LIN {X 0,Y 467.077,Z 400.09,A -85,B 0,C 180,E1 -7772.581,E2 -7772.581} C_VEL
LIN {X 0,Y 466.879,Z 403.998,A -85,B 0,C 180,E1 -7774.113,E2 -7774.113} C_VEL
LIN {X 0,Y 466.736,Z 406.492,A -85,B 0,C 180,E1 -7775.597,E2 -7775.597} C_VEL
LIN {X 0,Y 466.664,Z 407.771,A -85,B 0,C 180,E1 -7777.042,E2 -7777.042} C_VEL
LIN {X 0,Y 466.681,Z 407.948,A -85,B 0,C 180,E1 -7778.454,E2 -7778.454} C_VEL
LIN {X 0,Y 466.711,Z 407.112,A -85,B 0,C 180,E1 -7779.826,E2 -7779.826} C_VEL
LIN {X 0,Y 466.814,Z 404.771,A -85,B 0,C 180,E1 -7781.486,E2 -7781.486} C_VEL
LIN {X 0,Y 467.044,Z 400.686,A -85,B 0,C 180,E1 -7783.189,E2 -7783.189} C_VEL
LIN {X 0,Y 467.228,Z 395.648,A -85,B 0,C 180,E1 -7784.685,E2 -7784.685} C_VEL
LIN {X 0,Y 467.456,Z 388.922,A -85,B 0,C 180,E1 -7786.192,E2 -7786.192} C_VEL
LIN {X 0,Y 467.852,Z 381.695,A -85,B 0,C 180,E1 -7787.469,E2 -7787.469} C_VEL
LIN {X 0,Y 468.223,Z 373.379,A -85,B 0,C 180,E1 -7788.666,E2 -7788.666} C_VEL
LIN {X 0,Y 468.647,Z 364.557,A -85,B 0,C 180,E1 -7789.705,E2 -7789.705} C_VEL
LIN {X 0,Y 469.155,Z 353.711,A -85,B 0,C 180,E1 -7790.734,E2 -7790.734} C_VEL
LIN {X 0,Y 469.63,Z 342.193,A -85,B 0,C 180,E1 -7791.607,E2 -7791.607} C_VEL
LIN {X 0,Y 470.092,Z 330.037,A -85,B 0,C 180,E1 -7792.316,E2 -7792.316} C_VEL
LIN {X 0,Y 470.223,Z 319.07,A -85,B 0,C 180,E1 -7792.805,E2 -7792.805} C_VEL
LIN {X 0,Y 466.983,Z 306.035,A -85,B 0,C 180,E1 -7793.324,E2 -7793.324} C_VEL
LIN {X 0,Y 466.864,Z 305.117,A -85,B 0,C 180,E1 -7793.38,E2 -7793.38} C_VEL
LIN {X 0,Y 466.879,Z 302.169,A -85,B 0,C 180,E1 -7796.153,E2 -7796.153} C_VEL
LIN {X 0,Y 466.906,Z 298.871,A -85,B 0,C 180,E1 -7799.302,E2 -7799.302} C_VEL
LIN {X 0,Y 466.963,Z 296.873,A -85,B 0,C 180,E1 -7801.209,E2 -7801.209} C_VEL
LIN {X 0,Y 467.055,Z 296.311,A -85,B 0,C 180,E1 -7802.598,E2 -7802.598} C_VEL
LIN {X 0,Y 467.101,Z 296.304,A -85,B 0,C 180,E1 -7803.04,E2 -7803.04} C_VEL
LIN {X 0,Y 466.541,Z 296.375,A -85,B 0,C 180,E1 -7803.76,E2 -7803.76} C_VEL
LIN {X 0,Y 463.844,Z 296.712,A -85,B 0,C 180,E1 -7804.934,E2 -7804.934} C_VEL
LIN {X 0,Y 461.52,Z 297,A -85,B 0,C 180,E1 -7805.88,E2 -7805.88} C_VEL
LIN {X 0,Y 460.523,Z 297.122,A -85,B 0,C 180,E1 -7806.609,E2 -7806.609} C_VEL
LIN {X 0,Y 460.446,Z 297.13,A -85,B 0,C 180,E1 -7806.856,E2 -7806.856} C_VEL
LIN {X 0,Y 460.552,Z 297.12,A -85,B 0,C 180,E1 -7809.453,E2 -7809.453} C_VEL
LIN {X 0,Y 460.549,Z 297.118,A -85,B 0,C 180,E1 -7812.23,E2 -7812.23} C_VEL
LIN {X 0,Y 460.566,Z 297.118,A -85,B 0,C 180,E1 -7814.965,E2 -7814.965} C_VEL
LIN {X 0,Y 460.611,Z 297.11,A -85,B 0,C 180,E1 -7818.559,E2 -7818.559} C_VEL
LIN {X 0,Y 460.668,Z 297.101,A -85,B 0,C 180,E1 -7822.108,E2 -7822.108} C_VEL
LIN {X 0,Y 460.691,Z 297.101,A -85,B 0,C 180,E1 -7824.748,E2 -7824.748} C_VEL
LIN {X 0,Y 460.801,Z 297.086,A -85,B 0,C 180,E1 -7827.377,E2 -7827.377} C_VEL
LIN {X 0,Y 460.854,Z 297.078,A -85,B 0,C 180,E1 -7830,E2 -7830} C_VEL
LIN {X 0,Y 460.826,Z 297.084,A -85,B 0,C 180,E1 -7832.622,E2 -7832.622} C_VEL
LIN {X 0,Y 460.685,Z 297.102,A -85,B 0,C 180,E1 -7836.13,E2 -7836.13} C_VEL
LIN {X 0,Y 460.628,Z 297.109,A -85,B 0,C 180,E1 -7838.776,E2 -7838.776} C_VEL
LIN {X 0,Y 460.615,Z 297.112,A -85,B 0,C 180,E1 -7842.445,E2 -7842.445} C_VEL
LIN {X 0,Y 460.602,Z 297.111,A -85,B 0,C 180,E1 -7845.998,E2 -7845.998} C_VEL
LIN {X 0,Y 460.569,Z 297.114,A -85,B 0,C 180,E1 -7849.616,E2 -7849.616} C_VEL
LIN {X 0,Y 460.513,Z 297.123,A -85,B 0,C 180,E1 -7852.429,E2 -7852.429} C_VEL
LIN {X 0,Y 460.57,Z 297.117,A -85,B 0,C 180,E1 -7855.802,E2 -7855.802} C_VEL
LIN {X 0,Y 460.552,Z 297.119,A -85,B 0,C 180,E1 -7858.233,E2 -7858.233} C_VEL
LIN {X 0,Y 460.521,Z 297.12,A -85,B 0,C 180,E1 -7861.283,E2 -7861.283} C_VEL
LIN {X 0,Y 460.525,Z 297.122,A -85,B 0,C 180,E1 -7864.504,E2 -7864.504} C_VEL
LIN {X 0,Y 460.503,Z 297.125,A -85,B 0,C 180,E1 -7867.623,E2 -7867.623} C_VEL
LIN {X 0,Y 460.544,Z 297.119,A -85,B 0,C 180,E1 -7870.27,E2 -7870.27} C_VEL
LIN {X 0,Y 460.498,Z 297.124,A -85,B 0,C 180,E1 -7873.376,E2 -7873.376} C_VEL
LIN {X 0,Y 460.501,Z 297.123,A -85,B 0,C 180,E1 -7876.625,E2 -7876.625} C_VEL
LIN {X 0,Y 460.545,Z 297.119,A -85,B 0,C 180,E1 -7879.731,E2 -7879.731} C_VEL
LIN {X 0,Y 460.503,Z 297.123,A -85,B 0,C 180,E1 -7882.524,E2 -7882.524} C_VEL
LIN {X 0,Y 460.54,Z 297.122,A -85,B 0,C 180,E1 -7885.623,E2 -7885.623} C_VEL
LIN {X 0,Y 460.54,Z 297.119,A -85,B 0,C 180,E1 -7888.745,E2 -7888.745} C_VEL
LIN {X 0,Y 460.581,Z 297.114,A -85,B 0,C 180,E1 -7892.255,E2 -7892.255} C_VEL
LIN {X 0,Y 460.529,Z 297.121,A -85,B 0,C 180,E1 -7895.667,E2 -7895.667} C_VEL
LIN {X 0,Y 460.525,Z 297.12,A -85,B 0,C 180,E1 -7898.578,E2 -7898.578} C_VEL
LIN {X 0,Y 460.59,Z 297.115,A -85,B 0,C 180,E1 -7901.311,E2 -7901.311} C_VEL
LIN {X 0,Y 460.609,Z 297.11,A -85,B 0,C 180,E1 -7904.059,E2 -7904.059} C_VEL
LIN {X 0,Y 460.614,Z 297.111,A -85,B 0,C 180,E1 -7907.666,E2 -7907.666} C_VEL
LIN {X 0,Y 460.624,Z 297.109,A -85,B 0,C 180,E1 -7911.224,E2 -7911.224} C_VEL
LIN {X 0,Y 460.712,Z 297.096,A -85,B 0,C 180,E1 -7913.87,E2 -7913.87} C_VEL
LIN {X 0,Y 460.798,Z 297.087,A -85,B 0,C 180,E1 -7917.378,E2 -7917.378} C_VEL
LIN {X 0,Y 460.857,Z 297.079,A -85,B 0,C 180,E1 -7920,E2 -7920} C_VEL
LIN {X 0,Y 460.793,Z 297.09,A -85,B 0,C 180,E1 -7922.623,E2 -7922.623} C_VEL
LIN {X 0,Y 460.688,Z 297.1,A -85,B 0,C 180,E1 -7926.13,E2 -7926.13} C_VEL
LIN {X 0,Y 460.623,Z 297.11,A -85,B 0,C 180,E1 -7928.776,E2 -7928.776} C_VEL
LIN {X 0,Y 460.619,Z 297.11,A -85,B 0,C 180,E1 -7932.445,E2 -7932.445} C_VEL
LIN {X 0,Y 460.605,Z 297.111,A -85,B 0,C 180,E1 -7935.998,E2 -7935.998} C_VEL
LIN {X 0,Y 460.572,Z 297.115,A -85,B 0,C 180,E1 -7939.616,E2 -7939.616} C_VEL
LIN {X 0,Y 460.515,Z 297.123,A -85,B 0,C 180,E1 -7942.429,E2 -7942.429} C_VEL
LIN {X 0,Y 460.552,Z 297.117,A -85,B 0,C 180,E1 -7945.797,E2 -7945.797} C_VEL
LIN {X 0,Y 460.531,Z 297.121,A -85,B 0,C 180,E1 -7948.235,E2 -7948.235} C_VEL
LIN {X 0,Y 460.525,Z 297.121,A -85,B 0,C 180,E1 -7951.283,E2 -7951.283} C_VEL
LIN {X 0,Y 460.535,Z 297.12,A -85,B 0,C 180,E1 -7954.505,E2 -7954.505} C_VEL
LIN {X 0,Y 460.505,Z 297.123,A -85,B 0,C 180,E1 -7957.623,E2 -7957.623} C_VEL
LIN {X 0,Y 460.54,Z 297.121,A -85,B 0,C 180,E1 -7960.268,E2 -7960.268} C_VEL
LIN {X 0,Y 460.512,Z 297.124,A -85,B 0,C 180,E1 -7963.374,E2 -7963.374} C_VEL
LIN {X 0,Y 460.512,Z 297.121,A -85,B 0,C 180,E1 -7966.626,E2 -7966.626} C_VEL
LIN {X 0,Y 460.571,Z 297.238,A -85,B 0,C 180,E1 -7969.444,E2 -7969.444} C_VEL
LIN {X 0,Y 462.242,Z 306.265,A -85,B 0,C 180,E1 -7973.089,E2 -7973.089} C_VEL
LIN {X 0,Y 462.399,Z 310.595,A -85,B 0,C 180,E1 -7974.72,E2 -7974.72} C_VEL
LIN {X 0,Y 461.883,Z 319.246,A -85,B 0,C 180,E1 -7977.821,E2 -7977.821} C_VEL
LIN {X 0,Y 461.323,Z 329.384,A -85,B 0,C 180,E1 -7981.322,E2 -7981.322} C_VEL
LIN {X 0,Y 460.86,Z 339.544,A -85,B 0,C 180,E1 -7984.723,E2 -7984.723} C_VEL
LIN {X 0,Y 460.428,Z 349.692,A -85,B 0,C 180,E1 -7988.039,E2 -7988.039} C_VEL
LIN {X 0,Y 460.203,Z 359.887,A -85,B 0,C 180,E1 -7991.294,E2 -7991.294} C_VEL
LIN {X 0,Y 459.948,Z 369.672,A -85,B 0,C 180,E1 -7994.36,E2 -7994.36} C_VEL
LIN {X 0,Y 461.927,Z 384.605,A -85,B 0,C 180,E1 -7994.838,E2 -7994.838} C_VEL
LIN {X 0,Y 462.821,Z 394.468,A -85,B 0,C 180,E1 -7995.265,E2 -7995.265} C_VEL
LIN {X 0,Y 462.305,Z 406.889,A -85,B 0,C 180,E1 -7995.922,E2 -7995.922} C_VEL
LIN {X 0,Y 461.662,Z 419.477,A -85,B 0,C 180,E1 -7996.8,E2 -7996.8} C_VEL
LIN {X 0,Y 461.143,Z 430.593,A -85,B 0,C 180,E1 -7997.792,E2 -7997.792} C_VEL
LIN {X 0,Y 460.751,Z 439.624,A -85,B 0,C 180,E1 -7998.786,E2 -7998.786} C_VEL
LIN {X 0,Y 460.265,Z 449.421,A -85,B 0,C 180,E1 -8000.109,E2 -8000.109} C_VEL
LIN {X 0,Y 459.999,Z 457.267,A -85,B 0,C 180,E1 -8001.433,E2 -8001.433} C_VEL
LIN {X 0,Y 459.777,Z 464.466,A -85,B 0,C 180,E1 -8002.976,E2 -8002.976} C_VEL
LIN {X 0,Y 459.718,Z 469.266,A -85,B 0,C 180,E1 -8004.297,E2 -8004.297} C_VEL
LIN {X 0,Y 459.604,Z 472.924,A -85,B 0,C 180,E1 -8005.615,E2 -8005.615} C_VEL
LIN {X 0,Y 459.686,Z 474.819,A -85,B 0,C 180,E1 -8006.494,E2 -8006.494} C_VEL
LIN {X 0,Y 459.689,Z 476.233,A -85,B 0,C 180,E1 -8007.371,E2 -8007.371} C_VEL
LIN {X 0,Y 459.637,Z 477.228,A -85,B 0,C 180,E1 -8008.248,E2 -8008.248} C_VEL
LIN {X 0,Y 459.554,Z 478.027,A -85,B 0,C 180,E1 -8010,E2 -8010} C_VEL
LIN {X 0,Y 459.567,Z 477.788,A -85,B 0,C 180,E1 -8010.876,E2 -8010.876} C_VEL
LIN {X 0,Y 459.638,Z 477.151,A -85,B 0,C 180,E1 -8011.752,E2 -8011.752} C_VEL
LIN {X 0,Y 459.705,Z 476.116,A -85,B 0,C 180,E1 -8012.629,E2 -8012.629} C_VEL
LIN {X 0,Y 459.699,Z 474.666,A -85,B 0,C 180,E1 -8013.506,E2 -8013.506} C_VEL
LIN {X 0,Y 459.637,Z 471.625,A -85,B 0,C 180,E1 -8014.824,E2 -8014.824} C_VEL
LIN {X 0,Y 459.699,Z 467.531,A -85,B 0,C 180,E1 -8016.144,E2 -8016.144} C_VEL
LIN {X 0,Y 459.865,Z 461.251,A -85,B 0,C 180,E1 -8017.685,E2 -8017.685} C_VEL
LIN {X 0,Y 460.063,Z 454.403,A -85,B 0,C 180,E1 -8019.009,E2 -8019.009} C_VEL
LIN {X 0,Y 460.383,Z 445.938,A -85,B 0,C 180,E1 -8020.333,E2 -8020.333} C_VEL
LIN {X 0,Y 460.854,Z 437.273,A -85,B 0,C 180,E1 -8021.435,E2 -8021.435} C_VEL
LIN {X 0,Y 461.274,Z 427.652,A -85,B 0,C 180,E1 -8022.441,E2 -8022.441} C_VEL
LIN {X 0,Y 461.754,Z 416.085,A -85,B 0,C 180,E1 -8023.421,E2 -8023.421} C_VEL
LIN {X 0,Y 462.357,Z 404.606,A -85,B 0,C 180,E1 -8024.188,E2 -8024.188} C_VEL
LIN {X 0,Y 462.843,Z 392.852,A -85,B 0,C 180,E1 -8024.791,E2 -8024.791} C_VEL
LIN {X 0,Y 461.404,Z 379.556,A -85,B 0,C 180,E1 -8025.344,E2 -8025.344} C_VEL
LIN {X 0,Y 459.918,Z 368.362,A -85,B 0,C 180,E1 -8025.697,E2 -8025.697} C_VEL
LIN {X 0,Y 460.106,Z 358.542,A -85,B 0,C 180,E1 -8028.731,E2 -8028.731} C_VEL
LIN {X 0,Y 460.328,Z 349.752,A -85,B 0,C 180,E1 -8031.495,E2 -8031.495} C_VEL
LIN {X 0,Y 460.62,Z 339.486,A -85,B 0,C 180,E1 -8034.809,E2 -8034.809} C_VEL
LIN {X 0,Y 461.018,Z 330.389,A -85,B 0,C 180,E1 -8037.848,E2 -8037.848} C_VEL
LIN {X 0,Y 461.574,Z 319.93,A -85,B 0,C 180,E1 -8041.497,E2 -8041.497} C_VEL
LIN {X 0,Y 462.185,Z 311,A -85,B 0,C 180,E1 -8044.802,E2 -8044.802} C_VEL
LIN {X 0,Y 462.234,Z 307.021,A -85,B 0,C 180,E1 -8046.369,E2 -8046.369} C_VEL
LIN {X 0,Y 461.377,Z 301.675,A -85,B 0,C 180,E1 -8048.649,E2 -8048.649} C_VEL
LIN {X 0,Y 460.566,Z 297.118,A -85,B 0,C 180,E1 -8050.808,E2 -8050.808} C_VEL
LIN {X 0,Y 460.516,Z 297.127,A -85,B 0,C 180,E1 -8054.17,E2 -8054.17} C_VEL
LIN {X 0,Y 460.517,Z 297.127,A -85,B 0,C 180,E1 -8057.1,E2 -8057.1} C_VEL
LIN {X 0,Y 460.537,Z 297.123,A -85,B 0,C 180,E1 -8060.138,E2 -8060.138} C_VEL
LIN {X 0,Y 460.481,Z 297.127,A -85,B 0,C 180,E1 -8063.471,E2 -8063.471} C_VEL
LIN {X 0,Y 460.534,Z 297.121,A -85,B 0,C 180,E1 -8066.675,E2 -8066.675} C_VEL
LIN {X 0,Y 460.516,Z 297.123,A -85,B 0,C 180,E1 -8069.76,E2 -8069.76} C_VEL
LIN {X 0,Y 460.584,Z 297.114,A -85,B 0,C 180,E1 -8072.757,E2 -8072.757} C_VEL
LIN {X 0,Y 460.547,Z 297.117,A -85,B 0,C 180,E1 -8075.668,E2 -8075.668} C_VEL
LIN {X 0,Y 460.526,Z 297.122,A -85,B 0,C 180,E1 -8078.578,E2 -8078.578} C_VEL
LIN {X 0,Y 460.591,Z 297.114,A -85,B 0,C 180,E1 -8081.311,E2 -8081.311} C_VEL
LIN {X 0,Y 460.609,Z 297.111,A -85,B 0,C 180,E1 -8084.059,E2 -8084.059} C_VEL
LIN {X 0,Y 460.615,Z 297.111,A -85,B 0,C 180,E1 -8087.666,E2 -8087.666} C_VEL
LIN {X 0,Y 460.624,Z 297.109,A -85,B 0,C 180,E1 -8091.224,E2 -8091.224} C_VEL
LIN {X 0,Y 460.688,Z 297.101,A -85,B 0,C 180,E1 -8093.87,E2 -8093.87} C_VEL
LIN {X 0,Y 460.805,Z 297.087,A -85,B 0,C 180,E1 -8097.377,E2 -8097.377} C_VEL
LIN {X 0,Y 460.859,Z 297.082,A -85,B 0,C 180,E1 -8100,E2 -8100} C_VEL
LIN {X 0,Y 460.83,Z 297.084,A -85,B 0,C 180,E1 -8102.622,E2 -8102.622} C_VEL
LIN {X 0,Y 460.691,Z 297.103,A -85,B 0,C 180,E1 -8106.13,E2 -8106.13} C_VEL
LIN {X 0,Y 460.567,Z 297.118,A -85,B 0,C 180,E1 -8108.777,E2 -8108.777} C_VEL
LIN {X 0,Y 460.334,Z 297.148,A -85,B 0,C 180,E1 -8111.448,E2 -8111.448} C_VEL
LIN {X 0,Y 460.26,Z 297.442,A -85,B 0,C 180,E1 -8112.344,E2 -8112.344} C_VEL
LIN {X 0,Y 460.14,Z 300.675,A -85,B 0,C 180,E1 -8115.794,E2 -8115.794} C_VEL
LIN {X 0,Y 460.01,Z 303.468,A -85,B 0,C 180,E1 -8118.713,E2 -8118.713} C_VEL
LIN {X 0,Y 459.961,Z 306.142,A -85,B 0,C 180,E1 -8121.513,E2 -8121.513} C_VEL
LIN {X 0,Y 459.936,Z 307.052,A -85,B 0,C 180,E1 -8122.458,E2 -8122.458} C_VEL
LIN {X 0,Y 463.555,Z 320.766,A -85,B 0,C 180,E1 -8123.038,E2 -8123.038} C_VEL
LIN {X 0,Y 463.367,Z 332.506,A -85,B 0,C 180,E1 -8123.58,E2 -8123.58} C_VEL
LIN {X 0,Y 462.938,Z 343.442,A -85,B 0,C 180,E1 -8124.24,E2 -8124.24} C_VEL
LIN {X 0,Y 462.404,Z 354.286,A -85,B 0,C 180,E1 -8125.071,E2 -8125.071} C_VEL
LIN {X 0,Y 461.861,Z 365.295,A -85,B 0,C 180,E1 -8126.13,E2 -8126.13} C_VEL
LIN {X 0,Y 461.396,Z 374.199,A -85,B 0,C 180,E1 -8127.191,E2 -8127.191} C_VEL
LIN {X 0,Y 460.985,Z 382.758,A -85,B 0,C 180,E1 -8128.452,E2 -8128.452} C_VEL
LIN {X 0,Y 460.529,Z 390.5,A -85,B 0,C 180,E1 -8129.87,E2 -8129.87} C_VEL
LIN {X 0,Y 460.249,Z 396.54,A -85,B 0,C 180,E1 -8131.277,E2 -8131.277} C_VEL
LIN {X 0,Y 459.98,Z 401.571,A -85,B 0,C 180,E1 -8132.823,E2 -8132.823} C_VEL
LIN {X 0,Y 459.778,Z 405.325,A -85,B 0,C 180,E1 -8134.442,E2 -8134.442} C_VEL
LIN {X 0,Y 459.63,Z 407.418,A -85,B 0,C 180,E1 -8135.864,E2 -8135.864} C_VEL
LIN {X 0,Y 459.584,Z 408.46,A -85,B 0,C 180,E1 -8137.326,E2 -8137.326} C_VEL
LIN {X 0,Y 459.622,Z 408.377,A -85,B 0,C 180,E1 -8138.823,E2 -8138.823} C_VEL
LIN {X 0,Y 459.64,Z 407.369,A -85,B 0,C 180,E1 -8140.136,E2 -8140.136} C_VEL
LIN {X 0,Y 459.755,Z 405.367,A -85,B 0,C 180,E1 -8141.493,E2 -8141.493} C_VEL
LIN {X 0,Y 459.925,Z 402.426,A -85,B 0,C 180,E1 -8142.821,E2 -8142.821} C_VEL
LIN {X 0,Y 460.064,Z 398.573,A -85,B 0,C 180,E1 -8144.112,E2 -8144.112} C_VEL
LIN {X 0,Y 460.33,Z 392.861,A -85,B 0,C 180,E1 -8145.58,E2 -8145.58} C_VEL
LIN {X 0,Y 460.653,Z 385.313,A -85,B 0,C 180,E1 -8147.081,E2 -8147.081} C_VEL
LIN {X 0,Y 461.073,Z 377.507,A -85,B 0,C 180,E1 -8148.322,E2 -8148.322} C_VEL
LIN {X 0,Y 461.504,Z 369.477,A -85,B 0,C 180,E1 -8149.37,E2 -8149.37} C_VEL
LIN {X 0,Y 462.003,Z 359.381,A -85,B 0,C 180,E1 -8150.446,E2 -8150.446} C_VEL
LIN {X 0,Y 462.448,Z 349.392,A -85,B 0,C 180,E1 -8151.311,E2 -8151.311} C_VEL
LIN {X 0,Y 462.977,Z 337.6,A -85,B 0,C 180,E1 -8152.126,E2 -8152.126} C_VEL
LIN {X 0,Y 463.387,Z 326.476,A -85,B 0,C 180,E1 -8152.719,E2 -8152.719} C_VEL
LIN {X 0,Y 463.353,Z 320.314,A -85,B 0,C 180,E1 -8152.989,E2 -8152.989} C_VEL
LIN {X 0,Y 460.088,Z 307.047,A -85,B 0,C 180,E1 -8153.532,E2 -8153.532} C_VEL
LIN {X 0,Y 459.793,Z 305.583,A -85,B 0,C 180,E1 -8153.602,E2 -8153.602} C_VEL
LIN {X 0,Y 459.829,Z 301.774,A -85,B 0,C 180,E1 -8157.205,E2 -8157.205} C_VEL
LIN {X 0,Y 459.862,Z 298.238,A -85,B 0,C 180,E1 -8160.589,E2 -8160.589} C_VEL
LIN {X 0,Y 459.918,Z 297.202,A -85,B 0,C 180,E1 -8161.724,E2 -8161.724} C_VEL
LIN {X 0,Y 460.274,Z 297.154,A -85,B 0,C 180,E1 -8164.688,E2 -8164.688} C_VEL
LIN {X 0,Y 460.446,Z 297.13,A -85,B 0,C 180,E1 -8166.856,E2 -8166.856} C_VEL
LIN {X 0,Y 459.791,Z 297.213,A -85,B 0,C 180,E1 -8167.586,E2 -8167.586} C_VEL
LIN {X 0,Y 456.961,Z 297.565,A -85,B 0,C 180,E1 -8168.773,E2 -8168.773} C_VEL
LIN {X 0,Y 454.577,Z 297.861,A -85,B 0,C 180,E1 -8169.73,E2 -8169.73} C_VEL
LIN {X 0,Y 453.574,Z 297.985,A -85,B 0,C 180,E1 -8170.47,E2 -8170.47} C_VEL
LIN {X 0,Y 453.503,Z 297.995,A -85,B 0,C 180,E1 -8170.72,E2 -8170.72} C_VEL
LIN {X 0,Y 453.57,Z 297.985,A -85,B 0,C 180,E1 -8173.88,E2 -8173.88} C_VEL
LIN {X 0,Y 453.565,Z 297.988,A -85,B 0,C 180,E1 -8177.471,E2 -8177.471} C_VEL
LIN {X 0,Y 453.592,Z 297.986,A -85,B 0,C 180,E1 -8181.087,E2 -8181.087} C_VEL
LIN {X 0,Y 453.652,Z 297.977,A -85,B 0,C 180,E1 -8183.774,E2 -8183.774} C_VEL
LIN {X 0,Y 453.745,Z 297.965,A -85,B 0,C 180,E1 -8187.337,E2 -8187.337} C_VEL
LIN {X 0,Y 453.824,Z 297.954,A -85,B 0,C 180,E1 -8190,E2 -8190} C_VEL
LIN {X 0,Y 453.767,Z 297.963,A -85,B 0,C 180,E1 -8192.663,E2 -8192.663} C_VEL
LIN {X 0,Y 453.651,Z 297.978,A -85,B 0,C 180,E1 -8196.226,E2 -8196.226} C_VEL
LIN {X 0,Y 453.592,Z 297.985,A -85,B 0,C 180,E1 -8198.913,E2 -8198.913} C_VEL
LIN {X 0,Y 453.565,Z 297.99,A -85,B 0,C 180,E1 -8202.529,E2 -8202.529} C_VEL
LIN {X 0,Y 453.545,Z 297.992,A -85,B 0,C 180,E1 -8206.196,E2 -8206.196} C_VEL
LIN {X 0,Y 453.517,Z 297.993,A -85,B 0,C 180,E1 -8209.039,E2 -8209.039} C_VEL
LIN {X 0,Y 453.478,Z 298,A -85,B 0,C 180,E1 -8211.836,E2 -8211.836} C_VEL
LIN {X 0,Y 453.516,Z 297.993,A -85,B 0,C 180,E1 -8214.735,E2 -8214.735} C_VEL
LIN {X 0,Y 453.533,Z 297.993,A -85,B 0,C 180,E1 -8217.96,E2 -8217.96} C_VEL
LIN {X 0,Y 453.466,Z 297.999,A -85,B 0,C 180,E1 -8221.525,E2 -8221.525} C_VEL
LIN {X 0,Y 453.484,Z 297.998,A -85,B 0,C 180,E1 -8224.777,E2 -8224.777} C_VEL
LIN {X 0,Y 453.467,Z 298.002,A -85,B 0,C 180,E1 -8228.312,E2 -8228.312} C_VEL
LIN {X 0,Y 453.496,Z 297.996,A -85,B 0,C 180,E1 -8230.609,E2 -8230.609} C_VEL
LIN {X 0,Y 453.455,Z 298.001,A -85,B 0,C 180,E1 -8233.244,E2 -8233.244} C_VEL
LIN {X 0,Y 453.466,Z 298.001,A -85,B 0,C 180,E1 -8235.779,E2 -8235.779} C_VEL
LIN {X 0,Y 453.482,Z 297.998,A -85,B 0,C 180,E1 -8238.21,E2 -8238.21} C_VEL
LIN {X 0,Y 453.518,Z 297.993,A -85,B 0,C 180,E1 -8240.79,E2 -8240.79} C_VEL
LIN {X 0,Y 453.457,Z 298.002,A -85,B 0,C 180,E1 -8243.917,E2 -8243.917} C_VEL
LIN {X 0,Y 453.482,Z 298,A -85,B 0,C 180,E1 -8247.151,E2 -8247.151} C_VEL
LIN {X 0,Y 453.478,Z 297.997,A -85,B 0,C 180,E1 -8250.269,E2 -8250.269} C_VEL
LIN {X 0,Y 453.492,Z 297.998,A -85,B 0,C 180,E1 -8253.293,E2 -8253.293} C_VEL
LIN {X 0,Y 453.498,Z 297.996,A -85,B 0,C 180,E1 -8256.239,E2 -8256.239} C_VEL
LIN {X 0,Y 453.487,Z 297.999,A -85,B 0,C 180,E1 -8259.118,E2 -8259.118} C_VEL
LIN {X 0,Y 453.507,Z 297.994,A -85,B 0,C 180,E1 -8261.944,E2 -8261.944} C_VEL
LIN {X 0,Y 453.544,Z 297.99,A -85,B 0,C 180,E1 -8264.727,E2 -8264.727} C_VEL
LIN {X 0,Y 453.564,Z 297.988,A -85,B 0,C 180,E1 -8268.379,E2 -8268.379} C_VEL
LIN {X 0,Y 453.59,Z 297.986,A -85,B 0,C 180,E1 -8271.087,E2 -8271.087} C_VEL
LIN {X 0,Y 453.678,Z 297.972,A -85,B 0,C 180,E1 -8273.775,E2 -8273.775} C_VEL
LIN {X 0,Y 453.741,Z 297.966,A -85,B 0,C 180,E1 -8277.337,E2 -8277.337} C_VEL
LIN {X 0,Y 453.826,Z 297.955,A -85,B 0,C 180,E1 -8280,E2 -8280} C_VEL
LIN {X 0,Y 453.737,Z 297.968,A -85,B 0,C 180,E1 -8282.663,E2 -8282.663} C_VEL
LIN {X 0,Y 453.654,Z 297.976,A -85,B 0,C 180,E1 -8286.226,E2 -8286.226} C_VEL
LIN {X 0,Y 453.589,Z 297.987,A -85,B 0,C 180,E1 -8288.914,E2 -8288.914} C_VEL
LIN {X 0,Y 453.569,Z 297.988,A -85,B 0,C 180,E1 -8292.529,E2 -8292.529} C_VEL
LIN {X 0,Y 453.549,Z 297.99,A -85,B 0,C 180,E1 -8296.196,E2 -8296.196} C_VEL
LIN {X 0,Y 453.521,Z 297.994,A -85,B 0,C 180,E1 -8299.039,E2 -8299.039} C_VEL
LIN {X 0,Y 453.481,Z 297.997,A -85,B 0,C 180,E1 -8301.836,E2 -8301.836} C_VEL
LIN {X 0,Y 453.504,Z 297.996,A -85,B 0,C 180,E1 -8304.735,E2 -8304.735} C_VEL
LIN {X 0,Y 453.51,Z 297.995,A -85,B 0,C 180,E1 -8307.953,E2 -8307.953} C_VEL
LIN {X 0,Y 453.479,Z 297.999,A -85,B 0,C 180,E1 -8310.759,E2 -8310.759} C_VEL
LIN {X 0,Y 453.481,Z 298,A -85,B 0,C 180,E1 -8313.913,E2 -8313.913} C_VEL
LIN {X 0,Y 453.456,Z 297.999,A -85,B 0,C 180,E1 -8317.19,E2 -8317.19} C_VEL
LIN {X 0,Y 453.497,Z 297.999,A -85,B 0,C 180,E1 -8320.609,E2 -8320.609} C_VEL
LIN {X 0,Y 453.464,Z 298.003,A -85,B 0,C 180,E1 -8324.222,E2 -8324.222} C_VEL
LIN {X 0,Y 453.451,Z 298.001,A -85,B 0,C 180,E1 -8327.003,E2 -8327.003} C_VEL
LIN {X 0,Y 453.524,Z 298.12,A -85,B 0,C 180,E1 -8329.175,E2 -8329.175} C_VEL
LIN {X 0,Y 454.999,Z 306.165,A -85,B 0,C 180,E1 -8332.499,E2 -8332.499} C_VEL
LIN {X 0,Y 455.458,Z 310.258,A -85,B 0,C 180,E1 -8334.1,E2 -8334.1} C_VEL
LIN {X 0,Y 455.038,Z 317.82,A -85,B 0,C 180,E1 -8336.887,E2 -8336.887} C_VEL
LIN {X 0,Y 454.419,Z 327.55,A -85,B 0,C 180,E1 -8340.336,E2 -8340.336} C_VEL
LIN {X 0,Y 453.97,Z 336.21,A -85,B 0,C 180,E1 -8343.323,E2 -8343.323} C_VEL
LIN {X 0,Y 453.56,Z 344.906,A -85,B 0,C 180,E1 -8346.242,E2 -8346.242} C_VEL
LIN {X 0,Y 453.231,Z 355.085,A -85,B 0,C 180,E1 -8349.58,E2 -8349.58} C_VEL
LIN {X 0,Y 452.98,Z 365.211,A -85,B 0,C 180,E1 -8352.855,E2 -8352.855} C_VEL
LIN {X 0,Y 452.891,Z 369.199,A -85,B 0,C 180,E1 -8354.128,E2 -8354.128} C_VEL
LIN {X 0,Y 454.777,Z 383.374,A -85,B 0,C 180,E1 -8354.58,E2 -8354.58} C_VEL
LIN {X 0,Y 455.894,Z 394.935,A -85,B 0,C 180,E1 -8355.093,E2 -8355.093} C_VEL
LIN {X 0,Y 455.307,Z 407.962,A -85,B 0,C 180,E1 -8355.816,E2 -8355.816} C_VEL
LIN {X 0,Y 454.648,Z 420.017,A -85,B 0,C 180,E1 -8356.689,E2 -8356.689} C_VEL
LIN {X 0,Y 454.1,Z 431.05,A -85,B 0,C 180,E1 -8357.713,E2 -8357.713} C_VEL
LIN {X 0,Y 453.64,Z 440.82,A -85,B 0,C 180,E1 -8358.834,E2 -8358.834} C_VEL
LIN {X 0,Y 453.206,Z 448.837,A -85,B 0,C 180,E1 -8359.953,E2 -8359.953} C_VEL
LIN {X 0,Y 452.941,Z 456.702,A -85,B 0,C 180,E1 -8361.299,E2 -8361.299} C_VEL
LIN {X 0,Y 452.719,Z 463.909,A -85,B 0,C 180,E1 -8362.866,E2 -8362.866} C_VEL
LIN {X 0,Y 452.616,Z 468.714,A -85,B 0,C 180,E1 -8364.207,E2 -8364.207} C_VEL
LIN {X 0,Y 452.521,Z 472.38,A -85,B 0,C 180,E1 -8365.546,E2 -8365.546} C_VEL
LIN {X 0,Y 452.598,Z 474.277,A -85,B 0,C 180,E1 -8366.439,E2 -8366.439} C_VEL
LIN {X 0,Y 452.608,Z 475.696,A -85,B 0,C 180,E1 -8367.33,E2 -8367.33} C_VEL
LIN {X 0,Y 452.577,Z 476.693,A -85,B 0,C 180,E1 -8368.22,E2 -8368.22} C_VEL
LIN {X 0,Y 452.487,Z 477.491,A -85,B 0,C 180,E1 -8370,E2 -8370} C_VEL
LIN {X 0,Y 452.502,Z 477.254,A -85,B 0,C 180,E1 -8370.89,E2 -8370.89} C_VEL
LIN {X 0,Y 452.578,Z 476.615,A -85,B 0,C 180,E1 -8371.78,E2 -8371.78} C_VEL
LIN {X 0,Y 452.622,Z 475.576,A -85,B 0,C 180,E1 -8372.67,E2 -8372.67} C_VEL
LIN {X 0,Y 452.611,Z 474.124,A -85,B 0,C 180,E1 -8373.561,E2 -8373.561} C_VEL
LIN {X 0,Y 452.571,Z 471.082,A -85,B 0,C 180,E1 -8374.9,E2 -8374.9} C_VEL
LIN {X 0,Y 452.629,Z 466.354,A -85,B 0,C 180,E1 -8376.416,E2 -8376.416} C_VEL
LIN {X 0,Y 452.778,Z 460.702,A -85,B 0,C 180,E1 -8377.806,E2 -8377.806} C_VEL
LIN {X 0,Y 453.016,Z 453.859,A -85,B 0,C 180,E1 -8379.15,E2 -8379.15} C_VEL
LIN {X 0,Y 453.336,Z 445.389,A -85,B 0,C 180,E1 -8380.496,E2 -8380.496} C_VEL
LIN {X 0,Y 453.844,Z 436.728,A -85,B 0,C 180,E1 -8381.614,E2 -8381.614} C_VEL
LIN {X 0,Y 454.318,Z 426.807,A -85,B 0,C 180,E1 -8382.665,E2 -8382.665} C_VEL
LIN {X 0,Y 454.816,Z 415.576,A -85,B 0,C 180,E1 -8383.63,E2 -8383.63} C_VEL
LIN {X 0,Y 455.447,Z 404.137,A -85,B 0,C 180,E1 -8384.408,E2 -8384.408} C_VEL
LIN {X 0,Y 455.789,Z 392.449,A -85,B 0,C 180,E1 -8385.025,E2 -8385.025} C_VEL
LIN {X 0,Y 454.32,Z 378.63,A -85,B 0,C 180,E1 -8385.611,E2 -8385.611} C_VEL
LIN {X 0,Y 452.862,Z 367.781,A -85,B 0,C 180,E1 -8385.955,E2 -8385.955} C_VEL
LIN {X 0,Y 453.092,Z 356.616,A -85,B 0,C 180,E1 -8389.481,E2 -8389.481} C_VEL
LIN {X 0,Y 453.327,Z 347.819,A -85,B 0,C 180,E1 -8392.323,E2 -8392.323} C_VEL
LIN {X 0,Y 453.697,Z 337.61,A -85,B 0,C 180,E1 -8395.705,E2 -8395.705} C_VEL
LIN {X 0,Y 454.091,Z 328.971,A -85,B 0,C 180,E1 -8398.672,E2 -8398.672} C_VEL
LIN {X 0,Y 454.707,Z 319.141,A -85,B 0,C 180,E1 -8402.224,E2 -8402.224} C_VEL
LIN {X 0,Y 455.324,Z 310.676,A -85,B 0,C 180,E1 -8405.451,E2 -8405.451} C_VEL
LIN {X 0,Y 455.097,Z 306.862,A -85,B 0,C 180,E1 -8407.033,E2 -8407.033} C_VEL
LIN {X 0,Y 453.93,Z 300.307,A -85,B 0,C 180,E1 -8409.981,E2 -8409.981} C_VEL
LIN {X 0,Y 453.505,Z 297.997,A -85,B 0,C 180,E1 -8411.195,E2 -8411.195} C_VEL
LIN {X 0,Y 453.491,Z 298.001,A -85,B 0,C 180,E1 -8414.529,E2 -8414.529} C_VEL
LIN {X 0,Y 453.483,Z 298.003,A -85,B 0,C 180,E1 -8418.209,E2 -8418.209} C_VEL
LIN {X 0,Y 453.514,Z 297.999,A -85,B 0,C 180,E1 -8420.791,E2 -8420.791} C_VEL
LIN {X 0,Y 453.458,Z 298.002,A -85,B 0,C 180,E1 -8423.917,E2 -8423.917} C_VEL
LIN {X 0,Y 453.487,Z 298,A -85,B 0,C 180,E1 -8427.151,E2 -8427.151} C_VEL
LIN {X 0,Y 453.48,Z 298,A -85,B 0,C 180,E1 -8430.268,E2 -8430.268} C_VEL
LIN {X 0,Y 453.515,Z 297.996,A -85,B 0,C 180,E1 -8433.294,E2 -8433.294} C_VEL
LIN {X 0,Y 453.508,Z 297.997,A -85,B 0,C 180,E1 -8436.239,E2 -8436.239} C_VEL
LIN {X 0,Y 453.488,Z 298,A -85,B 0,C 180,E1 -8439.118,E2 -8439.118} C_VEL
LIN {X 0,Y 453.509,Z 297.995,A -85,B 0,C 180,E1 -8441.944,E2 -8441.944} C_VEL
LIN {X 0,Y 453.545,Z 297.989,A -85,B 0,C 180,E1 -8444.726,E2 -8444.726} C_VEL
LIN {X 0,Y 453.565,Z 297.988,A -85,B 0,C 180,E1 -8448.379,E2 -8448.379} C_VEL
LIN {X 0,Y 453.59,Z 297.985,A -85,B 0,C 180,E1 -8451.086,E2 -8451.086} C_VEL
LIN {X 0,Y 453.653,Z 297.977,A -85,B 0,C 180,E1 -8453.774,E2 -8453.774} C_VEL
LIN {X 0,Y 453.748,Z 297.966,A -85,B 0,C 180,E1 -8457.337,E2 -8457.337} C_VEL
LIN {X 0,Y 453.829,Z 297.957,A -85,B 0,C 180,E1 -8460,E2 -8460} C_VEL
LIN {X 0,Y 453.77,Z 297.964,A -85,B 0,C 180,E1 -8462.663,E2 -8462.663} C_VEL
LIN {X 0,Y 453.657,Z 297.979,A -85,B 0,C 180,E1 -8466.225,E2 -8466.225} C_VEL
LIN {X 0,Y 453.502,Z 297.999,A -85,B 0,C 180,E1 -8468.915,E2 -8468.915} C_VEL
LIN {X 0,Y 453.287,Z 298.025,A -85,B 0,C 180,E1 -8471.628,E2 -8471.628} C_VEL
LIN {X 0,Y 453.19,Z 298.529,A -85,B 0,C 180,E1 -8472.539,E2 -8472.539} C_VEL
LIN {X 0,Y 453.087,Z 301.68,A -85,B 0,C 180,E1 -8475.906,E2 -8475.906} C_VEL
LIN {X 0,Y 452.938,Z 304.62,A -85,B 0,C 180,E1 -8479.017,E2 -8479.017} C_VEL
LIN {X 0,Y 452.913,Z 307.675,A -85,B 0,C 180,E1 -8482.194,E2 -8482.194} C_VEL
LIN {X 0,Y 456.386,Z 320.769,A -85,B 0,C 180,E1 -8482.762,E2 -8482.762} C_VEL
LIN {X 0,Y 456.829,Z 322.748,A -85,B 0,C 180,E1 -8482.858,E2 -8482.858} C_VEL
LIN {X 0,Y 456.464,Z 335.298,A -85,B 0,C 180,E1 -8483.477,E2 -8483.477} C_VEL
LIN {X 0,Y 455.923,Z 346.924,A -85,B 0,C 180,E1 -8484.231,E2 -8484.231} C_VEL
LIN {X 0,Y 455.374,Z 357.66,A -85,B 0,C 180,E1 -8485.114,E2 -8485.114} C_VEL
LIN {X 0,Y 454.813,Z 368.325,A -85,B 0,C 180,E1 -8486.221,E2 -8486.221} C_VEL
LIN {X 0,Y 454.327,Z 377.499,A -85,B 0,C 180,E1 -8487.4,E2 -8487.4} C_VEL
LIN {X 0,Y 453.892,Z 385.609,A -85,B 0,C 180,E1 -8488.685,E2 -8488.685} C_VEL
LIN {X 0,Y 453.478,Z 392.222,A -85,B 0,C 180,E1 -8489.987,E2 -8489.987} C_VEL
LIN {X 0,Y 453.171,Z 398.151,A -85,B 0,C 180,E1 -8491.463,E2 -8491.463} C_VEL
LIN {X 0,Y 452.898,Z 403.043,A -85,B 0,C 180,E1 -8493.074,E2 -8493.074} C_VEL
LIN {X 0,Y 452.678,Z 406.312,A -85,B 0,C 180,E1 -8494.629,E2 -8494.629} C_VEL
LIN {X 0,Y 452.549,Z 408.284,A -85,B 0,C 180,E1 -8496.166,E2 -8496.166} C_VEL
LIN {X 0,Y 452.519,Z 409.054,A -85,B 0,C 180,E1 -8497.62,E2 -8497.62} C_VEL
LIN {X 0,Y 452.54,Z 408.781,A -85,B 0,C 180,E1 -8499.058,E2 -8499.058} C_VEL
LIN {X 0,Y 452.603,Z 407.205,A -85,B 0,C 180,E1 -8500.706,E2 -8500.706} C_VEL
LIN {X 0,Y 452.805,Z 403.952,A -85,B 0,C 180,E1 -8502.467,E2 -8502.467} C_VEL
LIN {X 0,Y 452.978,Z 400.724,A -85,B 0,C 180,E1 -8503.683,E2 -8503.683} C_VEL
LIN {X 0,Y 453.221,Z 395.29,A -85,B 0,C 180,E1 -8505.222,E2 -8505.222} C_VEL
LIN {X 0,Y 453.501,Z 388.312,A -85,B 0,C 180,E1 -8506.75,E2 -8506.75} C_VEL
LIN {X 0,Y 453.957,Z 381.119,A -85,B 0,C 180,E1 -8507.998,E2 -8507.998} C_VEL
LIN {X 0,Y 454.431,Z 372.044,A -85,B 0,C 180,E1 -8509.271,E2 -8509.271} C_VEL
LIN {X 0,Y 454.92,Z 362.567,A -85,B 0,C 180,E1 -8510.354,E2 -8510.354} C_VEL
LIN {X 0,Y 455.435,Z 352.171,A -85,B 0,C 180,E1 -8511.32,E2 -8511.32} C_VEL
LIN {X 0,Y 455.945,Z 340.997,A -85,B 0,C 180,E1 -8512.144,E2 -8512.144} C_VEL
LIN {X 0,Y 456.479,Z 327.793,A -85,B 0,C 180,E1 -8512.891,E2 -8512.891} C_VEL
LIN {X 0,Y 456.499,Z 321.537,A -85,B 0,C 180,E1 -8513.176,E2 -8513.176} C_VEL
LIN {X 0,Y 453.285,Z 308.554,A -85,B 0,C 180,E1 -8513.73,E2 -8513.73} C_VEL
LIN {X 0,Y 452.73,Z 306.066,A -85,B 0,C 180,E1 -8513.826,E2 -8513.826} C_VEL
LIN {X 0,Y 452.775,Z 302.604,A -85,B 0,C 180,E1 -8517.093,E2 -8517.093} C_VEL
LIN {X 0,Y 452.802,Z 299.195,A -85,B 0,C 180,E1 -8520.364,E2 -8520.364} C_VEL
LIN {X 0,Y 452.834,Z 298.286,A -85,B 0,C 180,E1 -8521.241,E2 -8521.241} C_VEL
LIN {X 0,Y 453.182,Z 298.035,A -85,B 0,C 180,E1 -8524.264,E2 -8524.264} C_VEL
LIN {X 0,Y 453.428,Z 298.006,A -85,B 0,C 180,E1 -8527.201,E2 -8527.201} C_VEL
LIN {X 0,Y 453.504,Z 297.993,A -85,B 0,C 180,E1 -8530.066,E2 -8530.066} C_VEL
LIN {X 0,Y 453.503,Z 297.995,A -85,B 0,C 180,E1 -8530.72,E2 -8530.72} C_VEL
LIN {X 0,Y 452.876,Z 298.078,A -85,B 0,C 180,E1 -8531.461,E2 -8531.461} C_VEL
LIN {X 0,Y 450.069,Z 298.429,A -85,B 0,C 180,E1 -8532.665,E2 -8532.665} C_VEL
LIN {X 0,Y 447.657,Z 298.726,A -85,B 0,C 180,E1 -8533.636,E2 -8533.636} C_VEL
LIN {X 0,Y 446.594,Z 298.855,A -85,B 0,C 180,E1 -8534.386,E2 -8534.386} C_VEL
LIN {X 0,Y 446.494,Z 298.867,A -85,B 0,C 180,E1 -8534.64,E2 -8534.64} C_VEL
LIN {X 0,Y 446.518,Z 298.864,A -85,B 0,C 180,E1 -8538.193,E2 -8538.193} C_VEL
LIN {X 0,Y 446.538,Z 298.864,A -85,B 0,C 180,E1 -8540.945,E2 -8540.945} C_VEL
LIN {X 0,Y 446.62,Z 298.853,A -85,B 0,C 180,E1 -8543.676,E2 -8543.676} C_VEL
LIN {X 0,Y 446.692,Z 298.844,A -85,B 0,C 180,E1 -8547.295,E2 -8547.295} C_VEL
LIN {X 0,Y 446.794,Z 298.829,A -85,B 0,C 180,E1 -8550,E2 -8550} C_VEL
LIN {X 0,Y 446.71,Z 298.843,A -85,B 0,C 180,E1 -8552.705,E2 -8552.705} C_VEL
LIN {X 0,Y 446.62,Z 298.854,A -85,B 0,C 180,E1 -8556.324,E2 -8556.324} C_VEL
LIN {X 0,Y 446.537,Z 298.863,A -85,B 0,C 180,E1 -8559.055,E2 -8559.055} C_VEL
LIN {X 0,Y 446.522,Z 298.866,A -85,B 0,C 180,E1 -8562.73,E2 -8562.73} C_VEL
LIN {X 0,Y 446.49,Z 298.871,A -85,B 0,C 180,E1 -8566.459,E2 -8566.459} C_VEL
LIN {X 0,Y 446.469,Z 298.87,A -85,B 0,C 180,E1 -8569.303,E2 -8569.303} C_VEL
LIN {X 0,Y 446.42,Z 298.879,A -85,B 0,C 180,E1 -8572.2,E2 -8572.2} C_VEL
LIN {X 0,Y 446.46,Z 298.872,A -85,B 0,C 180,E1 -8575.152,E2 -8575.152} C_VEL
LIN {X 0,Y 446.486,Z 298.872,A -85,B 0,C 180,E1 -8578.179,E2 -8578.179} C_VEL
LIN {X 0,Y 446.419,Z 298.878,A -85,B 0,C 180,E1 -8581.775,E2 -8581.775} C_VEL
LIN {X 0,Y 446.425,Z 298.878,A -85,B 0,C 180,E1 -8584.524,E2 -8584.524} C_VEL
LIN {X 0,Y 446.418,Z 298.879,A -85,B 0,C 180,E1 -8588.08,E2 -8588.08} C_VEL
LIN {X 0,Y 446.429,Z 298.876,A -85,B 0,C 180,E1 -8590.918,E2 -8590.918} C_VEL
LIN {X 0,Y 446.401,Z 298.883,A -85,B 0,C 180,E1 -8593.846,E2 -8593.846} C_VEL
LIN {X 0,Y 446.4,Z 298.881,A -85,B 0,C 180,E1 -8596.404,E2 -8596.404} C_VEL
LIN {X 0,Y 446.429,Z 298.876,A -85,B 0,C 180,E1 -8599.083,E2 -8599.083} C_VEL
LIN {X 0,Y 446.419,Z 298.879,A -85,B 0,C 180,E1 -8601.921,E2 -8601.921} C_VEL
LIN {X 0,Y 446.426,Z 298.878,A -85,B 0,C 180,E1 -8605.477,E2 -8605.477} C_VEL
LIN {X 0,Y 446.419,Z 298.877,A -85,B 0,C 180,E1 -8608.7,E2 -8608.7} C_VEL
LIN {X 0,Y 446.488,Z 298.871,A -85,B 0,C 180,E1 -8611.822,E2 -8611.822} C_VEL
LIN {X 0,Y 446.443,Z 298.875,A -85,B 0,C 180,E1 -8614.847,E2 -8614.847} C_VEL
LIN {X 0,Y 446.452,Z 298.872,A -85,B 0,C 180,E1 -8618.245,E2 -8618.245} C_VEL
LIN {X 0,Y 446.456,Z 298.873,A -85,B 0,C 180,E1 -8621.649,E2 -8621.649} C_VEL
LIN {X 0,Y 446.512,Z 298.866,A -85,B 0,C 180,E1 -8624.48,E2 -8624.48} C_VEL
LIN {X 0,Y 446.522,Z 298.865,A -85,B 0,C 180,E1 -8628.193,E2 -8628.193} C_VEL
LIN {X 0,Y 446.537,Z 298.865,A -85,B 0,C 180,E1 -8630.945,E2 -8630.945} C_VEL
LIN {X 0,Y 446.646,Z 298.848,A -85,B 0,C 180,E1 -8633.676,E2 -8633.676} C_VEL
LIN {X 0,Y 446.688,Z 298.845,A -85,B 0,C 180,E1 -8637.295,E2 -8637.295} C_VEL
LIN {X 0,Y 446.796,Z 298.831,A -85,B 0,C 180,E1 -8640,E2 -8640} C_VEL
LIN {X 0,Y 446.683,Z 298.847,A -85,B 0,C 180,E1 -8642.706,E2 -8642.706} C_VEL
LIN {X 0,Y 446.622,Z 298.853,A -85,B 0,C 180,E1 -8646.324,E2 -8646.324} C_VEL
LIN {X 0,Y 446.526,Z 298.863,A -85,B 0,C 180,E1 -8649.97,E2 -8649.97} C_VEL
LIN {X 0,Y 446.526,Z 298.867,A -85,B 0,C 180,E1 -8652.73,E2 -8652.73} C_VEL
LIN {X 0,Y 446.493,Z 298.87,A -85,B 0,C 180,E1 -8656.459,E2 -8656.459} C_VEL
LIN {X 0,Y 446.473,Z 298.871,A -85,B 0,C 180,E1 -8659.303,E2 -8659.303} C_VEL
LIN {X 0,Y 446.423,Z 298.88,A -85,B 0,C 180,E1 -8662.2,E2 -8662.2} C_VEL
LIN {X 0,Y 446.446,Z 298.872,A -85,B 0,C 180,E1 -8665.153,E2 -8665.153} C_VEL
LIN {X 0,Y 446.453,Z 298.874,A -85,B 0,C 180,E1 -8668.181,E2 -8668.181} C_VEL
LIN {X 0,Y 446.419,Z 298.877,A -85,B 0,C 180,E1 -8671.3,E2 -8671.3} C_VEL
LIN {X 0,Y 446.433,Z 298.876,A -85,B 0,C 180,E1 -8674.523,E2 -8674.523} C_VEL
LIN {X 0,Y 446.417,Z 298.88,A -85,B 0,C 180,E1 -8678.079,E2 -8678.079} C_VEL
LIN {X 0,Y 446.425,Z 298.877,A -85,B 0,C 180,E1 -8680.917,E2 -8680.917} C_VEL
LIN {X 0,Y 446.402,Z 298.881,A -85,B 0,C 180,E1 -8683.846,E2 -8683.846} C_VEL
LIN {X 0,Y 446.401,Z 298.879,A -85,B 0,C 180,E1 -8686.403,E2 -8686.403} C_VEL
LIN {X 0,Y 446.467,Z 298.943,A -85,B 0,C 180,E1 -8688.881,E2 -8688.881} C_VEL
LIN {X 0,Y 447.93,Z 306.999,A -85,B 0,C 180,E1 -8692.272,E2 -8692.272} C_VEL
LIN {X 0,Y 448.483,Z 311.336,A -85,B 0,C 180,E1 -8694.009,E2 -8694.009} C_VEL
LIN {X 0,Y 448.054,Z 318.524,A -85,B 0,C 180,E1 -8696.702,E2 -8696.702} C_VEL
LIN {X 0,Y 447.47,Z 327.161,A -85,B 0,C 180,E1 -8699.828,E2 -8699.828} C_VEL
LIN {X 0,Y 446.978,Z 335.801,A -85,B 0,C 180,E1 -8702.872,E2 -8702.872} C_VEL
LIN {X 0,Y 446.562,Z 344.64,A -85,B 0,C 180,E1 -8705.896,E2 -8705.896} C_VEL
LIN {X 0,Y 446.176,Z 354.594,A -85,B 0,C 180,E1 -8709.242,E2 -8709.242} C_VEL
LIN {X 0,Y 445.92,Z 364.722,A -85,B 0,C 180,E1 -8712.575,E2 -8712.575} C_VEL
LIN {X 0,Y 445.833,Z 368.844,A -85,B 0,C 180,E1 -8713.893,E2 -8713.893} C_VEL
LIN {X 0,Y 447.709,Z 382.921,A -85,B 0,C 180,E1 -8714.346,E2 -8714.346} C_VEL
LIN {X 0,Y 448.942,Z 395.301,A -85,B 0,C 180,E1 -8714.915,E2 -8714.915} C_VEL
LIN {X 0,Y 448.378,Z 407.251,A -85,B 0,C 180,E1 -8715.592,E2 -8715.592} C_VEL
LIN {X 0,Y 447.713,Z 419.325,A -85,B 0,C 180,E1 -8716.477,E2 -8716.477} C_VEL
LIN {X 0,Y 447.134,Z 430.411,A -85,B 0,C 180,E1 -8717.519,E2 -8717.519} C_VEL
LIN {X 0,Y 446.632,Z 440.197,A -85,B 0,C 180,E1 -8718.656,E2 -8718.656} C_VEL
LIN {X 0,Y 446.175,Z 448.231,A -85,B 0,C 180,E1 -8719.793,E2 -8719.793} C_VEL
LIN {X 0,Y 445.858,Z 456.115,A -85,B 0,C 180,E1 -8721.159,E2 -8721.159} C_VEL
LIN {X 0,Y 445.692,Z 461.482,A -85,B 0,C 180,E1 -8722.297,E2 -8722.297} C_VEL
LIN {X 0,Y 445.511,Z 467.503,A -85,B 0,C 180,E1 -8723.91,E2 -8723.91} C_VEL
LIN {X 0,Y 445.504,Z 470.749,A -85,B 0,C 180,E1 -8725.022,E2 -8725.022} C_VEL
LIN {X 0,Y 445.514,Z 473.73,A -85,B 0,C 180,E1 -8726.382,E2 -8726.382} C_VEL
LIN {X 0,Y 445.528,Z 475.154,A -85,B 0,C 180,E1 -8727.288,E2 -8727.288} C_VEL
LIN {X 0,Y 445.518,Z 476.155,A -85,B 0,C 180,E1 -8728.192,E2 -8728.192} C_VEL
LIN {X 0,Y 445.421,Z 476.956,A -85,B 0,C 180,E1 -8730,E2 -8730} C_VEL
LIN {X 0,Y 445.439,Z 476.721,A -85,B 0,C 180,E1 -8730.904,E2 -8730.904} C_VEL
LIN {X 0,Y 445.52,Z 476.083,A -85,B 0,C 180,E1 -8731.808,E2 -8731.808} C_VEL
LIN {X 0,Y 445.542,Z 475.041,A -85,B 0,C 180,E1 -8732.712,E2 -8732.712} C_VEL
LIN {X 0,Y 445.526,Z 473.588,A -85,B 0,C 180,E1 -8733.618,E2 -8733.618} C_VEL
LIN {X 0,Y 445.504,Z 470.545,A -85,B 0,C 180,E1 -8734.978,E2 -8734.978} C_VEL
LIN {X 0,Y 445.53,Z 466.29,A -85,B 0,C 180,E1 -8736.386,E2 -8736.386} C_VEL
LIN {X 0,Y 445.715,Z 460.162,A -85,B 0,C 180,E1 -8737.93,E2 -8737.93} C_VEL
LIN {X 0,Y 445.949,Z 453.32,A -85,B 0,C 180,E1 -8739.296,E2 -8739.296} C_VEL
LIN {X 0,Y 446.317,Z 444.86,A -85,B 0,C 180,E1 -8740.663,E2 -8740.663} C_VEL
LIN {X 0,Y 446.829,Z 436.212,A -85,B 0,C 180,E1 -8741.799,E2 -8741.799} C_VEL
LIN {X 0,Y 447.362,Z 425.658,A -85,B 0,C 180,E1 -8742.928,E2 -8742.928} C_VEL
LIN {X 0,Y 447.88,Z 415.091,A -85,B 0,C 180,E1 -8743.845,E2 -8743.845} C_VEL
LIN {X 0,Y 448.571,Z 403.708,A -85,B 0,C 180,E1 -8744.634,E2 -8744.634} C_VEL
LIN {X 0,Y 448.863,Z 393.331,A -85,B 0,C 180,E1 -8745.204,E2 -8745.204} C_VEL
LIN {X 0,Y 447.572,Z 380.4,A -85,B 0,C 180,E1 -8745.79,E2 -8745.79} C_VEL
LIN {X 0,Y 445.812,Z 367.183,A -85,B 0,C 180,E1 -8746.236,E2 -8746.236} C_VEL
LIN {X 0,Y 446.019,Z 356.125,A -85,B 0,C 180,E1 -8749.803,E2 -8749.803} C_VEL
LIN {X 0,Y 446.294,Z 347.363,A -85,B 0,C 180,E1 -8752.694,E2 -8752.694} C_VEL
LIN {X 0,Y 446.725,Z 336.844,A -85,B 0,C 180,E1 -8756.267,E2 -8756.267} C_VEL
LIN {X 0,Y 447.095,Z 328.661,A -85,B 0,C 180,E1 -8759.163,E2 -8759.163} C_VEL
LIN {X 0,Y 447.719,Z 320.256,A -85,B 0,C 180,E1 -8762.257,E2 -8762.257} C_VEL
LIN {X 0,Y 448.335,Z 312.049,A -85,B 0,C 180,E1 -8765.451,E2 -8765.451} C_VEL
LIN {X 0,Y 448.195,Z 308.598,A -85,B 0,C 180,E1 -8766.897,E2 -8766.897} C_VEL
LIN {X 0,Y 446.966,Z 301.542,A -85,B 0,C 180,E1 -8770.142,E2 -8770.142} C_VEL
LIN {X 0,Y 446.455,Z 298.875,A -85,B 0,C 180,E1 -8771.539,E2 -8771.539} C_VEL
LIN {X 0,Y 446.458,Z 298.88,A -85,B 0,C 180,E1 -8775.103,E2 -8775.103} C_VEL
LIN {X 0,Y 446.432,Z 298.88,A -85,B 0,C 180,E1 -8778.609,E2 -8778.609} C_VEL
LIN {X 0,Y 446.46,Z 298.878,A -85,B 0,C 180,E1 -8780.974,E2 -8780.974} C_VEL
LIN {X 0,Y 446.423,Z 298.879,A -85,B 0,C 180,E1 -8784.374,E2 -8784.374} C_VEL
LIN {X 0,Y 446.427,Z 298.878,A -85,B 0,C 180,E1 -8787.639,E2 -8787.639} C_VEL
LIN {X 0,Y 446.454,Z 298.875,A -85,B 0,C 180,E1 -8790.791,E2 -8790.791} C_VEL
LIN {X 0,Y 446.482,Z 298.871,A -85,B 0,C 180,E1 -8793.849,E2 -8793.849} C_VEL
LIN {X 0,Y 446.434,Z 298.878,A -85,B 0,C 180,E1 -8796.823,E2 -8796.823} C_VEL
LIN {X 0,Y 446.449,Z 298.874,A -85,B 0,C 180,E1 -8799.737,E2 -8799.737} C_VEL
LIN {X 0,Y 446.462,Z 298.872,A -85,B 0,C 180,E1 -8802.597,E2 -8802.597} C_VEL
LIN {X 0,Y 446.476,Z 298.872,A -85,B 0,C 180,E1 -8805.412,E2 -8805.412} C_VEL
LIN {X 0,Y 446.523,Z 298.867,A -85,B 0,C 180,E1 -8808.193,E2 -8808.193} C_VEL
LIN {X 0,Y 446.537,Z 298.864,A -85,B 0,C 180,E1 -8810.944,E2 -8810.944} C_VEL
LIN {X 0,Y 446.622,Z 298.853,A -85,B 0,C 180,E1 -8813.676,E2 -8813.676} C_VEL
LIN {X 0,Y 446.695,Z 298.844,A -85,B 0,C 180,E1 -8817.295,E2 -8817.295} C_VEL
LIN {X 0,Y 446.798,Z 298.833,A -85,B 0,C 180,E1 -8820,E2 -8820} C_VEL
LIN {X 0,Y 446.714,Z 298.843,A -85,B 0,C 180,E1 -8822.705,E2 -8822.705} C_VEL
LIN {X 0,Y 446.625,Z 298.855,A -85,B 0,C 180,E1 -8826.324,E2 -8826.324} C_VEL
LIN {X 0,Y 446.452,Z 298.877,A -85,B 0,C 180,E1 -8829.057,E2 -8829.057} C_VEL
LIN {X 0,Y 446.224,Z 298.905,A -85,B 0,C 180,E1 -8831.815,E2 -8831.815} C_VEL
LIN {X 0,Y 446.068,Z 302.224,A -85,B 0,C 180,E1 -8835.536,E2 -8835.536} C_VEL
LIN {X 0,Y 445.894,Z 305.44,A -85,B 0,C 180,E1 -8838.967,E2 -8838.967} C_VEL
LIN {X 0,Y 445.856,Z 308.239,A -85,B 0,C 180,E1 -8841.916,E2 -8841.916} C_VEL
LIN {X 0,Y 449.653,Z 322.166,A -85,B 0,C 180,E1 -8842.546,E2 -8842.546} C_VEL
LIN {X 0,Y 449.94,Z 326.44,A -85,B 0,C 180,E1 -8842.748,E2 -8842.748} C_VEL
LIN {X 0,Y 449.491,Z 339.25,A -85,B 0,C 180,E1 -8843.436,E2 -8843.436} C_VEL
LIN {X 0,Y 448.927,Z 351.441,A -85,B 0,C 180,E1 -8844.313,E2 -8844.313} C_VEL
LIN {X 0,Y 448.292,Z 362.201,A -85,B 0,C 180,E1 -8845.29,E2 -8845.29} C_VEL
LIN {X 0,Y 447.811,Z 371.085,A -85,B 0,C 180,E1 -8846.287,E2 -8846.287} C_VEL
LIN {X 0,Y 447.334,Z 378.989,A -85,B 0,C 180,E1 -8847.358,E2 -8847.358} C_VEL
LIN {X 0,Y 446.869,Z 387.061,A -85,B 0,C 180,E1 -8848.699,E2 -8848.699} C_VEL
LIN {X 0,Y 446.418,Z 393.495,A -85,B 0,C 180,E1 -8850.017,E2 -8850.017} C_VEL
LIN {X 0,Y 446.137,Z 398.602,A -85,B 0,C 180,E1 -8851.322,E2 -8851.322} C_VEL
LIN {X 0,Y 445.863,Z 403.262,A -85,B 0,C 180,E1 -8852.862,E2 -8852.862} C_VEL
LIN {X 0,Y 445.63,Z 406.902,A -85,B 0,C 180,E1 -8854.594,E2 -8854.594} C_VEL
LIN {X 0,Y 445.47,Z 409.077,A -85,B 0,C 180,E1 -8856.427,E2 -8856.427} C_VEL
LIN {X 0,Y 445.45,Z 409.641,A -85,B 0,C 180,E1 -8857.975,E2 -8857.975} C_VEL
LIN {X 0,Y 445.477,Z 409.14,A -85,B 0,C 180,E1 -8859.372,E2 -8859.372} C_VEL
LIN {X 0,Y 445.547,Z 407.67,A -85,B 0,C 180,E1 -8860.786,E2 -8860.786} C_VEL
LIN {X 0,Y 445.696,Z 405.254,A -85,B 0,C 180,E1 -8862.172,E2 -8862.172} C_VEL
LIN {X 0,Y 445.9,Z 401.9,A -85,B 0,C 180,E1 -8863.529,E2 -8863.529} C_VEL
LIN {X 0,Y 446.076,Z 397.623,A -85,B 0,C 180,E1 -8864.847,E2 -8864.847} C_VEL
LIN {X 0,Y 446.378,Z 391.121,A -85,B 0,C 180,E1 -8866.406,E2 -8866.406} C_VEL
LIN {X 0,Y 446.891,Z 382.884,A -85,B 0,C 180,E1 -8867.932,E2 -8867.932} C_VEL
LIN {X 0,Y 447.337,Z 374.802,A -85,B 0,C 180,E1 -8869.14,E2 -8869.14} C_VEL
LIN {X 0,Y 447.881,Z 364.861,A -85,B 0,C 180,E1 -8870.342,E2 -8870.342} C_VEL
LIN {X 0,Y 448.468,Z 353.845,A -85,B 0,C 180,E1 -8871.41,E2 -8871.41} C_VEL
LIN {X 0,Y 448.976,Z 343.21,A -85,B 0,C 180,E1 -8872.236,E2 -8872.236} C_VEL
LIN {X 0,Y 449.453,Z 332.565,A -85,B 0,C 180,E1 -8872.89,E2 -8872.89} C_VEL
LIN {X 0,Y 449.758,Z 324.234,A -85,B 0,C 180,E1 -8873.294,E2 -8873.294} C_VEL
LIN {X 0,Y 447.806,Z 315.127,A -85,B 0,C 180,E1 -8873.726,E2 -8873.726} C_VEL
LIN {X 0,Y 445.663,Z 306.527,A -85,B 0,C 180,E1 -8874.078,E2 -8874.078} C_VEL
LIN {X 0,Y 445.696,Z 302.825,A -85,B 0,C 180,E1 -8877.579,E2 -8877.579} C_VEL
LIN {X 0,Y 445.74,Z 299.533,A -85,B 0,C 180,E1 -8880.739,E2 -8880.739} C_VEL
LIN {X 0,Y 445.859,Z 298.952,A -85,B 0,C 180,E1 -8881.972,E2 -8881.972} C_VEL
LIN {X 0,Y 446.189,Z 298.908,A -85,B 0,C 180,E1 -8884.831,E2 -8884.831} C_VEL
LIN {X 0,Y 446.447,Z 298.874,A -85,B 0,C 180,E1 -8888.246,E2 -8888.246} C_VEL
LIN {X 0,Y 446.452,Z 298.874,A -85,B 0,C 180,E1 -8891.649,E2 -8891.649} C_VEL
LIN {X 0,Y 446.494,Z 298.867,A -85,B 0,C 180,E1 -8894.64,E2 -8894.64} C_VEL
LIN {X 0,Y 445.795,Z 298.956,A -85,B 0,C 180,E1 -8895.393,E2 -8895.393} C_VEL
LIN {X 0,Y 442.947,Z 299.311,A -85,B 0,C 180,E1 -8896.618,E2 -8896.618} C_VEL
LIN {X 0,Y 440.556,Z 299.607,A -85,B 0,C 180,E1 -8897.606,E2 -8897.606} C_VEL
LIN {X 0,Y 439.526,Z 299.735,A -85,B 0,C 180,E1 -8898.369,E2 -8898.369} C_VEL
LIN {X 0,Y 439.439,Z 299.746,A -85,B 0,C 180,E1 -8898.627,E2 -8898.627} C_VEL
LIN {X 0,Y 439.534,Z 299.734,A -85,B 0,C 180,E1 -8901.726,E2 -8901.726} C_VEL
LIN {X 0,Y 439.611,Z 299.727,A -85,B 0,C 180,E1 -8904.496,E2 -8904.496} C_VEL
LIN {X 0,Y 439.634,Z 299.723,A -85,B 0,C 180,E1 -8908.168,E2 -8908.168} C_VEL
LIN {X 0,Y 439.764,Z 299.705,A -85,B 0,C 180,E1 -8910,E2 -8910} C_VEL
LIN {X 0,Y 439.657,Z 299.721,A -85,B 0,C 180,E1 -8912.749,E2 -8912.749} C_VEL
LIN {X 0,Y 439.592,Z 299.729,A -85,B 0,C 180,E1 -8916.426,E2 -8916.426} C_VEL
LIN {X 0,Y 439.499,Z 299.74,A -85,B 0,C 180,E1 -8919.202,E2 -8919.202} C_VEL
LIN {X 0,Y 439.466,Z 299.744,A -85,B 0,C 180,E1 -8922.938,E2 -8922.938} C_VEL
LIN {X 0,Y 439.447,Z 299.749,A -85,B 0,C 180,E1 -8926.348,E2 -8926.348} C_VEL
LIN {X 0,Y 439.403,Z 299.751,A -85,B 0,C 180,E1 -8929.626,E2 -8929.626} C_VEL
LIN {X 0,Y 439.367,Z 299.758,A -85,B 0,C 180,E1 -8932.576,E2 -8932.576} C_VEL
LIN {X 0,Y 439.407,Z 299.751,A -85,B 0,C 180,E1 -8935.585,E2 -8935.585} C_VEL
LIN {X 0,Y 439.418,Z 299.75,A -85,B 0,C 180,E1 -8938.674,E2 -8938.674} C_VEL
LIN {X 0,Y 439.37,Z 299.758,A -85,B 0,C 180,E1 -8942.03,E2 -8942.03} C_VEL
LIN {X 0,Y 439.394,Z 299.752,A -85,B 0,C 180,E1 -8945.34,E2 -8945.34} C_VEL
LIN {X 0,Y 439.38,Z 299.754,A -85,B 0,C 180,E1 -8948.596,E2 -8948.596} C_VEL
LIN {X 0,Y 439.39,Z 299.753,A -85,B 0,C 180,E1 -8951.257,E2 -8951.257} C_VEL
LIN {X 0,Y 439.401,Z 299.751,A -85,B 0,C 180,E1 -8954.73,E2 -8954.73} C_VEL
LIN {X 0,Y 439.398,Z 299.755,A -85,B 0,C 180,E1 -8957.796,E2 -8957.796} C_VEL
LIN {X 0,Y 439.439,Z 299.748,A -85,B 0,C 180,E1 -8960.229,E2 -8960.229} C_VEL
LIN {X 0,Y 439.376,Z 299.756,A -85,B 0,C 180,E1 -8963.713,E2 -8963.713} C_VEL
LIN {X 0,Y 439.375,Z 299.756,A -85,B 0,C 180,E1 -8967.054,E2 -8967.054} C_VEL
LIN {X 0,Y 439.385,Z 299.753,A -85,B 0,C 180,E1 -8970.274,E2 -8970.274} C_VEL
LIN {X 0,Y 439.422,Z 299.751,A -85,B 0,C 180,E1 -8973.396,E2 -8973.396} C_VEL
LIN {X 0,Y 439.386,Z 299.753,A -85,B 0,C 180,E1 -8976.43,E2 -8976.43} C_VEL
LIN {X 0,Y 439.393,Z 299.754,A -85,B 0,C 180,E1 -8979.397,E2 -8979.397} C_VEL
LIN {X 0,Y 439.41,Z 299.749,A -85,B 0,C 180,E1 -8982.309,E2 -8982.309} C_VEL
LIN {X 0,Y 439.452,Z 299.748,A -85,B 0,C 180,E1 -8985.174,E2 -8985.174} C_VEL
LIN {X 0,Y 439.488,Z 299.741,A -85,B 0,C 180,E1 -8988.002,E2 -8988.002} C_VEL
LIN {X 0,Y 439.508,Z 299.739,A -85,B 0,C 180,E1 -8991.726,E2 -8991.726} C_VEL
LIN {X 0,Y 439.623,Z 299.724,A -85,B 0,C 180,E1 -8994.496,E2 -8994.496} C_VEL
LIN {X 0,Y 439.638,Z 299.721,A -85,B 0,C 180,E1 -8998.168,E2 -8998.168} C_VEL
LIN {X 0,Y 439.766,Z 299.706,A -85,B 0,C 180,E1 -9000,E2 -9000} C_VEL
LIN {X 0,Y 439.633,Z 299.725,A -85,B 0,C 180,E1 -9002.749,E2 -9002.749} C_VEL
LIN {X 0,Y 439.594,Z 299.729,A -85,B 0,C 180,E1 -9006.426,E2 -9006.426} C_VEL
LIN {X 0,Y 439.5,Z 299.739,A -85,B 0,C 180,E1 -9009.202,E2 -9009.202} C_VEL
LIN {X 0,Y 439.47,Z 299.744,A -85,B 0,C 180,E1 -9012.938,E2 -9012.938} C_VEL
LIN {X 0,Y 439.451,Z 299.746,A -85,B 0,C 180,E1 -9016.348,E2 -9016.348} C_VEL
LIN {X 0,Y 439.406,Z 299.751,A -85,B 0,C 180,E1 -9019.626,E2 -9019.626} C_VEL
LIN {X 0,Y 439.368,Z 299.757,A -85,B 0,C 180,E1 -9022.575,E2 -9022.575} C_VEL
LIN {X 0,Y 439.384,Z 299.752,A -85,B 0,C 180,E1 -9025.586,E2 -9025.586} C_VEL
LIN {X 0,Y 439.404,Z 299.752,A -85,B 0,C 180,E1 -9028.675,E2 -9028.675} C_VEL
LIN {X 0,Y 439.374,Z 299.756,A -85,B 0,C 180,E1 -9032.03,E2 -9032.03} C_VEL
LIN {X 0,Y 439.398,Z 299.752,A -85,B 0,C 180,E1 -9035.34,E2 -9035.34} C_VEL
LIN {X 0,Y 439.374,Z 299.756,A -85,B 0,C 180,E1 -9038.596,E2 -9038.596} C_VEL
LIN {X 0,Y 439.385,Z 299.752,A -85,B 0,C 180,E1 -9041.256,E2 -9041.256} C_VEL
LIN {X 0,Y 439.402,Z 299.751,A -85,B 0,C 180,E1 -9044.729,E2 -9044.729} C_VEL
LIN {X 0,Y 439.412,Z 299.751,A -85,B 0,C 180,E1 -9048.563,E2 -9048.563} C_VEL
LIN {X 0,Y 440.642,Z 306.615,A -85,B 0,C 180,E1 -9051.535,E2 -9051.535} C_VEL
LIN {X 0,Y 441.398,Z 311.019,A -85,B 0,C 180,E1 -9053.36,E2 -9053.36} C_VEL
LIN {X 0,Y 441.35,Z 315.276,A -85,B 0,C 180,E1 -9055.022,E2 -9055.022} C_VEL
LIN {X 0,Y 440.723,Z 323.886,A -85,B 0,C 180,E1 -9058.248,E2 -9058.248} C_VEL
LIN {X 0,Y 440.193,Z 332.615,A -85,B 0,C 180,E1 -9061.416,E2 -9061.416} C_VEL
LIN {X 0,Y 439.65,Z 342.591,A -85,B 0,C 180,E1 -9064.937,E2 -9064.937} C_VEL
LIN {X 0,Y 439.172,Z 352.685,A -85,B 0,C 180,E1 -9068.403,E2 -9068.403} C_VEL
LIN {X 0,Y 438.904,Z 362.757,A -85,B 0,C 180,E1 -9071.805,E2 -9071.805} C_VEL
LIN {X 0,Y 438.768,Z 368.38,A -85,B 0,C 180,E1 -9073.643,E2 -9073.643} C_VEL
LIN {X 0,Y 440.631,Z 382.075,A -85,B 0,C 180,E1 -9074.093,E2 -9074.093} C_VEL
LIN {X 0,Y 441.915,Z 394.466,A -85,B 0,C 180,E1 -9074.669,E2 -9074.669} C_VEL
LIN {X 0,Y 441.464,Z 406.493,A -85,B 0,C 180,E1 -9075.361,E2 -9075.361} C_VEL
LIN {X 0,Y 440.754,Z 418.66,A -85,B 0,C 180,E1 -9076.263,E2 -9076.263} C_VEL
LIN {X 0,Y 440.157,Z 429.747,A -85,B 0,C 180,E1 -9077.318,E2 -9077.318} C_VEL
LIN {X 0,Y 439.634,Z 439.561,A -85,B 0,C 180,E1 -9078.473,E2 -9078.473} C_VEL
LIN {X 0,Y 439.153,Z 447.616,A -85,B 0,C 180,E1 -9079.628,E2 -9079.628} C_VEL
LIN {X 0,Y 438.793,Z 455.525,A -85,B 0,C 180,E1 -9081.016,E2 -9081.016} C_VEL
LIN {X 0,Y 438.604,Z 460.899,A -85,B 0,C 180,E1 -9082.172,E2 -9082.172} C_VEL
LIN {X 0,Y 438.449,Z 466.356,A -85,B 0,C 180,E1 -9083.625,E2 -9083.625} C_VEL
LIN {X 0,Y 438.439,Z 470.194,A -85,B 0,C 180,E1 -9084.942,E2 -9084.942} C_VEL
LIN {X 0,Y 438.416,Z 473.178,A -85,B 0,C 180,E1 -9086.324,E2 -9086.324} C_VEL
LIN {X 0,Y 438.452,Z 474.611,A -85,B 0,C 180,E1 -9087.244,E2 -9087.244} C_VEL
LIN {X 0,Y 438.46,Z 475.615,A -85,B 0,C 180,E1 -9088.163,E2 -9088.163} C_VEL
LIN {X 0,Y 438.358,Z 476.419,A -85,B 0,C 180,E1 -9090,E2 -9090} C_VEL
LIN {X 0,Y 438.378,Z 476.188,A -85,B 0,C 180,E1 -9090.919,E2 -9090.919} C_VEL
LIN {X 0,Y 438.462,Z 475.549,A -85,B 0,C 180,E1 -9091.837,E2 -9091.837} C_VEL
LIN {X 0,Y 438.465,Z 474.507,A -85,B 0,C 180,E1 -9092.756,E2 -9092.756} C_VEL
LIN {X 0,Y 438.428,Z 473.053,A -85,B 0,C 180,E1 -9093.676,E2 -9093.676} C_VEL
LIN {X 0,Y 438.437,Z 470.012,A -85,B 0,C 180,E1 -9095.058,E2 -9095.058} C_VEL
LIN {X 0,Y 438.466,Z 465.913,A -85,B 0,C 180,E1 -9096.442,E2 -9096.442} C_VEL
LIN {X 0,Y 438.662,Z 459.638,A -85,B 0,C 180,E1 -9098.059,E2 -9098.059} C_VEL
LIN {X 0,Y 438.884,Z 452.794,A -85,B 0,C 180,E1 -9099.447,E2 -9099.447} C_VEL
LIN {X 0,Y 439.315,Z 444.345,A -85,B 0,C 180,E1 -9100.835,E2 -9100.835} C_VEL
LIN {X 0,Y 439.818,Z 435.72,A -85,B 0,C 180,E1 -9101.99,E2 -9101.99} C_VEL
LIN {X 0,Y 440.381,Z 425.171,A -85,B 0,C 180,E1 -9103.139,E2 -9103.139} C_VEL
LIN {X 0,Y 440.991,Z 414.684,A -85,B 0,C 180,E1 -9104.066,E2 -9104.066} C_VEL
LIN {X 0,Y 441.7,Z 403.349,A -85,B 0,C 180,E1 -9104.867,E2 -9104.867} C_VEL
LIN {X 0,Y 441.942,Z 394.148,A -85,B 0,C 180,E1 -9105.389,E2 -9105.389} C_VEL
LIN {X 0,Y 440.727,Z 380.971,A -85,B 0,C 180,E1 -9106.019,E2 -9106.019} C_VEL
LIN {X 0,Y 438.915,Z 368.213,A -85,B 0,C 180,E1 -9106.466,E2 -9106.466} C_VEL
LIN {X 0,Y 438.758,Z 366.617,A -85,B 0,C 180,E1 -9106.515,E2 -9106.515} C_VEL
LIN {X 0,Y 438.963,Z 355.634,A -85,B 0,C 180,E1 -9110.135,E2 -9110.135} C_VEL
LIN {X 0,Y 439.265,Z 346.919,A -85,B 0,C 180,E1 -9113.078,E2 -9113.078} C_VEL
LIN {X 0,Y 439.709,Z 336.798,A -85,B 0,C 180,E1 -9116.586,E2 -9116.586} C_VEL
LIN {X 0,Y 440.14,Z 328.287,A -85,B 0,C 180,E1 -9119.67,E2 -9119.67} C_VEL
LIN {X 0,Y 440.772,Z 319.986,A -85,B 0,C 180,E1 -9122.829,E2 -9122.829} C_VEL
LIN {X 0,Y 441.394,Z 312.799,A -85,B 0,C 180,E1 -9125.704,E2 -9125.704} C_VEL
LIN {X 0,Y 441.112,Z 309.211,A -85,B 0,C 180,E1 -9127.26,E2 -9127.26} C_VEL
LIN {X 0,Y 440.111,Z 303.481,A -85,B 0,C 180,E1 -9129.959,E2 -9129.959} C_VEL
LIN {X 0,Y 439.395,Z 299.756,A -85,B 0,C 180,E1 -9131.954,E2 -9131.954} C_VEL
LIN {X 0,Y 439.405,Z 299.758,A -85,B 0,C 180,E1 -9135.271,E2 -9135.271} C_VEL
LIN {X 0,Y 439.392,Z 299.757,A -85,B 0,C 180,E1 -9138.743,E2 -9138.743} C_VEL
LIN {X 0,Y 439.381,Z 299.757,A -85,B 0,C 180,E1 -9141.607,E2 -9141.607} C_VEL
LIN {X 0,Y 439.403,Z 299.753,A -85,B 0,C 180,E1 -9144.844,E2 -9144.844} C_VEL
LIN {X 0,Y 439.378,Z 299.757,A -85,B 0,C 180,E1 -9148.14,E2 -9148.14} C_VEL
LIN {X 0,Y 439.437,Z 299.748,A -85,B 0,C 180,E1 -9151.598,E2 -9151.598} C_VEL
LIN {X 0,Y 439.41,Z 299.752,A -85,B 0,C 180,E1 -9154.415,E2 -9154.415} C_VEL
LIN {X 0,Y 439.37,Z 299.755,A -85,B 0,C 180,E1 -9157.425,E2 -9157.425} C_VEL
LIN {X 0,Y 439.446,Z 299.747,A -85,B 0,C 180,E1 -9160.663,E2 -9160.663} C_VEL
LIN {X 0,Y 439.468,Z 299.743,A -85,B 0,C 180,E1 -9164.225,E2 -9164.225} C_VEL
LIN {X 0,Y 439.489,Z 299.744,A -85,B 0,C 180,E1 -9168.001,E2 -9168.001} C_VEL
LIN {X 0,Y 439.508,Z 299.739,A -85,B 0,C 180,E1 -9171.725,E2 -9171.725} C_VEL
LIN {X 0,Y 439.613,Z 299.727,A -85,B 0,C 180,E1 -9174.496,E2 -9174.496} C_VEL
LIN {X 0,Y 439.639,Z 299.725,A -85,B 0,C 180,E1 -9178.168,E2 -9178.168} C_VEL
LIN {X 0,Y 439.768,Z 299.709,A -85,B 0,C 180,E1 -9180,E2 -9180} C_VEL
LIN {X 0,Y 439.661,Z 299.721,A -85,B 0,C 180,E1 -9182.749,E2 -9182.749} C_VEL
LIN {X 0,Y 439.597,Z 299.73,A -85,B 0,C 180,E1 -9186.425,E2 -9186.425} C_VEL
LIN {X 0,Y 439.384,Z 299.758,A -85,B 0,C 180,E1 -9189.204,E2 -9189.204} C_VEL
LIN {X 0,Y 439.169,Z 299.917,A -85,B 0,C 180,E1 -9192.007,E2 -9192.007} C_VEL
LIN {X 0,Y 439.013,Z 303.384,A -85,B 0,C 180,E1 -9195.792,E2 -9195.792} C_VEL
LIN {X 0,Y 438.856,Z 306.467,A -85,B 0,C 180,E1 -9199.116,E2 -9199.116} C_VEL
LIN {X 0,Y 438.81,Z 308.814,A -85,B 0,C 180,E1 -9201.615,E2 -9201.615} C_VEL
LIN {X 0,Y 442.623,Z 322.786,A -85,B 0,C 180,E1 -9202.278,E2 -9202.278} C_VEL
LIN {X 0,Y 443.183,Z 325.951,A -85,B 0,C 180,E1 -9202.444,E2 -9202.444} C_VEL
LIN {X 0,Y 442.739,Z 338.877,A -85,B 0,C 180,E1 -9203.135,E2 -9203.135} C_VEL
LIN {X 0,Y 442.168,Z 349.943,A -85,B 0,C 180,E1 -9203.91,E2 -9203.91} C_VEL
LIN {X 0,Y 441.573,Z 360.788,A -85,B 0,C 180,E1 -9204.878,E2 -9204.878} C_VEL
LIN {X 0,Y 440.943,Z 370.904,A -85,B 0,C 180,E1 -9205.996,E2 -9205.996} C_VEL
LIN {X 0,Y 440.433,Z 378.989,A -85,B 0,C 180,E1 -9207.091,E2 -9207.091} C_VEL
LIN {X 0,Y 439.976,Z 386.281,A -85,B 0,C 180,E1 -9208.284,E2 -9208.284} C_VEL
LIN {X 0,Y 439.458,Z 393.392,A -85,B 0,C 180,E1 -9209.72,E2 -9209.72} C_VEL
LIN {X 0,Y 439.086,Z 399.646,A -85,B 0,C 180,E1 -9211.345,E2 -9211.345} C_VEL
LIN {X 0,Y 438.775,Z 404.391,A -85,B 0,C 180,E1 -9212.997,E2 -9212.997} C_VEL
LIN {X 0,Y 438.622,Z 406.724,A -85,B 0,C 180,E1 -9214.111,E2 -9214.111} C_VEL
LIN {X 0,Y 438.471,Z 408.478,A -85,B 0,C 180,E1 -9215.241,E2 -9215.241} C_VEL
LIN {X 0,Y 438.395,Z 409.827,A -85,B 0,C 180,E1 -9216.72,E2 -9216.72} C_VEL
LIN {X 0,Y 438.367,Z 410.144,A -85,B 0,C 180,E1 -9218.225,E2 -9218.225} C_VEL
LIN {X 0,Y 438.421,Z 409.258,A -85,B 0,C 180,E1 -9219.882,E2 -9219.882} C_VEL
LIN {X 0,Y 438.569,Z 406.844,A -85,B 0,C 180,E1 -9221.684,E2 -9221.684} C_VEL
LIN {X 0,Y 438.787,Z 404.06,A -85,B 0,C 180,E1 -9222.985,E2 -9222.985} C_VEL
LIN {X 0,Y 438.927,Z 400.325,A -85,B 0,C 180,E1 -9224.302,E2 -9224.302} C_VEL
LIN {X 0,Y 439.184,Z 395.618,A -85,B 0,C 180,E1 -9225.604,E2 -9225.604} C_VEL
LIN {X 0,Y 439.534,Z 388.714,A -85,B 0,C 180,E1 -9227.122,E2 -9227.122} C_VEL
LIN {X 0,Y 440.043,Z 380.765,A -85,B 0,C 180,E1 -9228.501,E2 -9228.501} C_VEL
LIN {X 0,Y 440.617,Z 371.437,A -85,B 0,C 180,E1 -9229.809,E2 -9229.809} C_VEL
LIN {X 0,Y 441.2,Z 361.97,A -85,B 0,C 180,E1 -9230.885,E2 -9230.885} C_VEL
LIN {X 0,Y 441.763,Z 350.859,A -85,B 0,C 180,E1 -9231.9,E2 -9231.9} C_VEL
LIN {X 0,Y 442.275,Z 339.969,A -85,B 0,C 180,E1 -9232.695,E2 -9232.695} C_VEL
LIN {X 0,Y 442.832,Z 327.815,A -85,B 0,C 180,E1 -9233.38,E2 -9233.38} C_VEL
LIN {X 0,Y 442.571,Z 323.088,A -85,B 0,C 180,E1 -9233.61,E2 -9233.61} C_VEL
LIN {X 0,Y 439.292,Z 309.938,A -85,B 0,C 180,E1 -9234.201,E2 -9234.201} C_VEL
LIN {X 0,Y 438.61,Z 306.999,A -85,B 0,C 180,E1 -9234.313,E2 -9234.313} C_VEL
LIN {X 0,Y 438.613,Z 304.192,A -85,B 0,C 180,E1 -9236.989,E2 -9236.989} C_VEL
LIN {X 0,Y 438.697,Z 300.807,A -85,B 0,C 180,E1 -9240.223,E2 -9240.223} C_VEL
LIN {X 0,Y 438.699,Z 299.845,A -85,B 0,C 180,E1 -9241.275,E2 -9241.275} C_VEL
LIN {X 0,Y 439.081,Z 299.792,A -85,B 0,C 180,E1 -9244.395,E2 -9244.395} C_VEL
LIN {X 0,Y 439.323,Z 299.762,A -85,B 0,C 180,E1 -9247.422,E2 -9247.422} C_VEL
LIN {X 0,Y 439.403,Z 299.75,A -85,B 0,C 180,E1 -9250.374,E2 -9250.374} C_VEL
LIN {X 0,Y 439.447,Z 299.746,A -85,B 0,C 180,E1 -9253.652,E2 -9253.652} C_VEL
LIN {X 0,Y 439.467,Z 299.745,A -85,B 0,C 180,E1 -9257.062,E2 -9257.062} C_VEL
LIN {X 0,Y 439.439,Z 299.746,A -85,B 0,C 180,E1 -9258.627,E2 -9258.627} C_VEL
LIN {X 0,Y 438.774,Z 299.834,A -85,B 0,C 180,E1 -9259.392,E2 -9259.392} C_VEL
LIN {X 0,Y 435.965,Z 300.186,A -85,B 0,C 180,E1 -9260.636,E2 -9260.636} C_VEL
LIN {X 0,Y 433.597,Z 300.479,A -85,B 0,C 180,E1 -9261.639,E2 -9261.639} C_VEL
LIN {X 0,Y 432.585,Z 300.602,A -85,B 0,C 180,E1 -9262.414,E2 -9262.414} C_VEL
LIN {X 0,Y 432.505,Z 300.61,A -85,B 0,C 180,E1 -9262.676,E2 -9262.676} C_VEL
LIN {X 0,Y 432.586,Z 300.602,A -85,B 0,C 180,E1 -9264.406,E2 -9264.406} C_VEL
LIN {X 0,Y 432.604,Z 300.599,A -85,B 0,C 180,E1 -9268.138,E2 -9268.138} C_VEL
LIN {X 0,Y 432.733,Z 300.581,A -85,B 0,C 180,E1 -9270,E2 -9270} C_VEL
LIN {X 0,Y 432.606,Z 300.6,A -85,B 0,C 180,E1 -9272.794,E2 -9272.794} C_VEL
LIN {X 0,Y 432.586,Z 300.6,A -85,B 0,C 180,E1 -9275.594,E2 -9275.594} C_VEL
LIN {X 0,Y 432.483,Z 300.616,A -85,B 0,C 180,E1 -9278.41,E2 -9278.41} C_VEL
LIN {X 0,Y 432.46,Z 300.617,A -85,B 0,C 180,E1 -9282.197,E2 -9282.197} C_VEL
LIN {X 0,Y 432.431,Z 300.62,A -85,B 0,C 180,E1 -9286.039,E2 -9286.039} C_VEL
LIN {X 0,Y 432.387,Z 300.624,A -85,B 0,C 180,E1 -9289.485,E2 -9289.485} C_VEL
LIN {X 0,Y 432.321,Z 300.633,A -85,B 0,C 180,E1 -9292.964,E2 -9292.964} C_VEL
LIN {X 0,Y 432.366,Z 300.629,A -85,B 0,C 180,E1 -9296.033,E2 -9296.033} C_VEL
LIN {X 0,Y 432.344,Z 300.63,A -85,B 0,C 180,E1 -9299.188,E2 -9299.188} C_VEL
LIN {X 0,Y 432.324,Z 300.634,A -85,B 0,C 180,E1 -9302.443,E2 -9302.443} C_VEL
LIN {X 0,Y 432.344,Z 300.631,A -85,B 0,C 180,E1 -9305.632,E2 -9305.632} C_VEL
LIN {X 0,Y 432.348,Z 300.63,A -85,B 0,C 180,E1 -9309.343,E2 -9309.343} C_VEL
LIN {X 0,Y 432.335,Z 300.633,A -85,B 0,C 180,E1 -9311.797,E2 -9311.797} C_VEL
LIN {X 0,Y 432.335,Z 300.632,A -85,B 0,C 180,E1 -9314.348,E2 -9314.348} C_VEL
LIN {X 0,Y 432.322,Z 300.633,A -85,B 0,C 180,E1 -9317.016,E2 -9317.016} C_VEL
LIN {X 0,Y 432.344,Z 300.632,A -85,B 0,C 180,E1 -9319.82,E2 -9319.82} C_VEL
LIN {X 0,Y 432.309,Z 300.635,A -85,B 0,C 180,E1 -9323.022,E2 -9323.022} C_VEL
LIN {X 0,Y 432.36,Z 300.629,A -85,B 0,C 180,E1 -9325.997,E2 -9325.997} C_VEL
LIN {X 0,Y 432.351,Z 300.632,A -85,B 0,C 180,E1 -9329.49,E2 -9329.49} C_VEL
LIN {X 0,Y 432.388,Z 300.625,A -85,B 0,C 180,E1 -9332.928,E2 -9332.928} C_VEL
LIN {X 0,Y 432.37,Z 300.628,A -85,B 0,C 180,E1 -9336.023,E2 -9336.023} C_VEL
LIN {X 0,Y 432.354,Z 300.632,A -85,B 0,C 180,E1 -9339.046,E2 -9339.046} C_VEL
LIN {X 0,Y 432.365,Z 300.627,A -85,B 0,C 180,E1 -9342.011,E2 -9342.011} C_VEL
LIN {X 0,Y 432.399,Z 300.625,A -85,B 0,C 180,E1 -9344.927,E2 -9344.927} C_VEL
LIN {X 0,Y 432.464,Z 300.616,A -85,B 0,C 180,E1 -9347.804,E2 -9347.804} C_VEL
LIN {X 0,Y 432.468,Z 300.616,A -85,B 0,C 180,E1 -9351.59,E2 -9351.59} C_VEL
LIN {X 0,Y 432.6,Z 300.598,A -85,B 0,C 180,E1 -9354.406,E2 -9354.406} C_VEL
LIN {X 0,Y 432.607,Z 300.596,A -85,B 0,C 180,E1 -9358.138,E2 -9358.138} C_VEL
LIN {X 0,Y 432.735,Z 300.582,A -85,B 0,C 180,E1 -9360,E2 -9360} C_VEL
LIN {X 0,Y 432.584,Z 300.603,A -85,B 0,C 180,E1 -9362.794,E2 -9362.794} C_VEL
LIN {X 0,Y 432.589,Z 300.598,A -85,B 0,C 180,E1 -9365.594,E2 -9365.594} C_VEL
LIN {X 0,Y 432.468,Z 300.616,A -85,B 0,C 180,E1 -9368.41,E2 -9368.41} C_VEL
LIN {X 0,Y 432.464,Z 300.617,A -85,B 0,C 180,E1 -9372.197,E2 -9372.197} C_VEL
LIN {X 0,Y 432.434,Z 300.621,A -85,B 0,C 180,E1 -9376.039,E2 -9376.039} C_VEL
LIN {X 0,Y 432.391,Z 300.624,A -85,B 0,C 180,E1 -9379.485,E2 -9379.485} C_VEL
LIN {X 0,Y 432.322,Z 300.635,A -85,B 0,C 180,E1 -9382.964,E2 -9382.964} C_VEL
LIN {X 0,Y 432.343,Z 300.63,A -85,B 0,C 180,E1 -9385.002,E2 -9385.002} C_VEL
LIN {X 0,Y 432.351,Z 300.631,A -85,B 0,C 180,E1 -9388.126,E2 -9388.126} C_VEL
LIN {X 0,Y 432.325,Z 300.633,A -85,B 0,C 180,E1 -9391.346,E2 -9391.346} C_VEL
LIN {X 0,Y 432.343,Z 300.632,A -85,B 0,C 180,E1 -9394.677,E2 -9394.677} C_VEL
LIN {X 0,Y 432.337,Z 300.633,A -85,B 0,C 180,E1 -9398.15,E2 -9398.15} C_VEL
LIN {X 0,Y 432.328,Z 300.633,A -85,B 0,C 180,E1 -9401.601,E2 -9401.601} C_VEL
LIN {X 0,Y 432.337,Z 300.633,A -85,B 0,C 180,E1 -9404.347,E2 -9404.347} C_VEL
LIN {X 0,Y 432.319,Z 300.633,A -85,B 0,C 180,E1 -9407.016,E2 -9407.016} C_VEL
LIN {X 0,Y 432.398,Z 300.839,A -85,B 0,C 180,E1 -9408.389,E2 -9408.389} C_VEL
LIN {X 0,Y 433.709,Z 308.045,A -85,B 0,C 180,E1 -9411.554,E2 -9411.554} C_VEL
LIN {X 0,Y 434.397,Z 312.015,A -85,B 0,C 180,E1 -9413.229,E2 -9413.229} C_VEL
LIN {X 0,Y 434.372,Z 316.322,A -85,B 0,C 180,E1 -9414.944,E2 -9414.944} C_VEL
LIN {X 0,Y 433.698,Z 324.917,A -85,B 0,C 180,E1 -9418.22,E2 -9418.22} C_VEL
LIN {X 0,Y 433.137,Z 333.914,A -85,B 0,C 180,E1 -9421.547,E2 -9421.547} C_VEL
LIN {X 0,Y 432.581,Z 343.591,A -85,B 0,C 180,E1 -9425.013,E2 -9425.013} C_VEL
LIN {X 0,Y 432.095,Z 353.639,A -85,B 0,C 180,E1 -9428.533,E2 -9428.533} C_VEL
LIN {X 0,Y 431.783,Z 363.686,A -85,B 0,C 180,E1 -9431.985,E2 -9431.985} C_VEL
LIN {X 0,Y 431.714,Z 367.824,A -85,B 0,C 180,E1 -9433.388,E2 -9433.388} C_VEL
LIN {X 0,Y 433.583,Z 382.051,A -85,B 0,C 180,E1 -9433.865,E2 -9433.865} C_VEL
LIN {X 0,Y 434.919,Z 394.728,A -85,B 0,C 180,E1 -9434.476,E2 -9434.476} C_VEL
LIN {X 0,Y 434.583,Z 405.723,A -85,B 0,C 180,E1 -9435.124,E2 -9435.124} C_VEL
LIN {X 0,Y 433.805,Z 418.217,A -85,B 0,C 180,E1 -9436.063,E2 -9436.063} C_VEL
LIN {X 0,Y 433.196,Z 429.068,A -85,B 0,C 180,E1 -9437.11,E2 -9437.11} C_VEL
LIN {X 0,Y 432.635,Z 438.905,A -85,B 0,C 180,E1 -9438.284,E2 -9438.284} C_VEL
LIN {X 0,Y 432.124,Z 446.981,A -85,B 0,C 180,E1 -9439.457,E2 -9439.457} C_VEL
LIN {X 0,Y 431.736,Z 454.917,A -85,B 0,C 180,E1 -9440.868,E2 -9440.868} C_VEL
LIN {X 0,Y 431.544,Z 460.301,A -85,B 0,C 180,E1 -9442.043,E2 -9442.043} C_VEL
LIN {X 0,Y 431.352,Z 466.194,A -85,B 0,C 180,E1 -9443.655,E2 -9443.655} C_VEL
LIN {X 0,Y 431.373,Z 469.627,A -85,B 0,C 180,E1 -9444.859,E2 -9444.859} C_VEL
LIN {X 0,Y 431.321,Z 472.618,A -85,B 0,C 180,E1 -9446.263,E2 -9446.263} C_VEL
LIN {X 0,Y 431.377,Z 474.063,A -85,B 0,C 180,E1 -9447.198,E2 -9447.198} C_VEL
LIN {X 0,Y 431.404,Z 475.072,A -85,B 0,C 180,E1 -9448.133,E2 -9448.133} C_VEL
LIN {X 0,Y 431.296,Z 475.882,A -85,B 0,C 180,E1 -9450,E2 -9450} C_VEL
LIN {X 0,Y 431.32,Z 475.657,A -85,B 0,C 180,E1 -9450.934,E2 -9450.934} C_VEL
LIN {X 0,Y 431.39,Z 475.019,A -85,B 0,C 180,E1 -9451.867,E2 -9451.867} C_VEL
LIN {X 0,Y 431.389,Z 473.975,A -85,B 0,C 180,E1 -9452.801,E2 -9452.801} C_VEL
LIN {X 0,Y 431.331,Z 472.521,A -85,B 0,C 180,E1 -9453.737,E2 -9453.737} C_VEL
LIN {X 0,Y 431.369,Z 469.483,A -85,B 0,C 180,E1 -9455.141,E2 -9455.141} C_VEL
LIN {X 0,Y 431.382,Z 465.388,A -85,B 0,C 180,E1 -9456.548,E2 -9456.548} C_VEL
LIN {X 0,Y 431.588,Z 459.126,A -85,B 0,C 180,E1 -9458.192,E2 -9458.192} C_VEL
LIN {X 0,Y 431.843,Z 452.298,A -85,B 0,C 180,E1 -9459.603,E2 -9459.603} C_VEL
LIN {X 0,Y 432.306,Z 443.862,A -85,B 0,C 180,E1 -9461.012,E2 -9461.012} C_VEL
LIN {X 0,Y 432.792,Z 435.254,A -85,B 0,C 180,E1 -9462.187,E2 -9462.187} C_VEL
LIN {X 0,Y 433.407,Z 424.7,A -85,B 0,C 180,E1 -9463.358,E2 -9463.358} C_VEL
LIN {X 0,Y 434.09,Z 414.277,A -85,B 0,C 180,E1 -9464.294,E2 -9464.294} C_VEL
LIN {X 0,Y 434.839,Z 402.988,A -85,B 0,C 180,E1 -9465.107,E2 -9465.107} C_VEL
LIN {X 0,Y 435.056,Z 394.967,A -85,B 0,C 180,E1 -9465.579,E2 -9465.579} C_VEL
LIN {X 0,Y 433.862,Z 381.481,A -85,B 0,C 180,E1 -9466.253,E2 -9466.253} C_VEL
LIN {X 0,Y 431.914,Z 367.85,A -85,B 0,C 180,E1 -9466.759,E2 -9466.759} C_VEL
LIN {X 0,Y 431.681,Z 365.962,A -85,B 0,C 180,E1 -9466.832,E2 -9466.832} C_VEL
LIN {X 0,Y 431.927,Z 355.154,A -85,B 0,C 180,E1 -9470.477,E2 -9470.477} C_VEL
LIN {X 0,Y 432.227,Z 346.474,A -85,B 0,C 180,E1 -9473.477,E2 -9473.477} C_VEL
LIN {X 0,Y 432.747,Z 336.467,A -85,B 0,C 180,E1 -9477.048,E2 -9477.048} C_VEL
LIN {X 0,Y 433.224,Z 328.022,A -85,B 0,C 180,E1 -9480.192,E2 -9480.192} C_VEL
LIN {X 0,Y 433.804,Z 320.902,A -85,B 0,C 180,E1 -9482.954,E2 -9482.954} C_VEL
LIN {X 0,Y 434.451,Z 313.428,A -85,B 0,C 180,E1 -9486.017,E2 -9486.017} C_VEL
LIN {X 0,Y 433.913,Z 309.073,A -85,B 0,C 180,E1 -9487.987,E2 -9487.987} C_VEL
LIN {X 0,Y 432.806,Z 302.849,A -85,B 0,C 180,E1 -9491.058,E2 -9491.058} C_VEL
LIN {X 0,Y 432.375,Z 300.629,A -85,B 0,C 180,E1 -9492.263,E2 -9492.263} C_VEL
LIN {X 0,Y 432.337,Z 300.638,A -85,B 0,C 180,E1 -9495.665,E2 -9495.665} C_VEL
LIN {X 0,Y 432.337,Z 300.636,A -85,B 0,C 180,E1 -9498.398,E2 -9498.398} C_VEL
LIN {X 0,Y 432.343,Z 300.633,A -85,B 0,C 180,E1 -9501.85,E2 -9501.85} C_VEL
LIN {X 0,Y 432.344,Z 300.631,A -85,B 0,C 180,E1 -9505.323,E2 -9505.323} C_VEL
LIN {X 0,Y 432.326,Z 300.634,A -85,B 0,C 180,E1 -9508.654,E2 -9508.654} C_VEL
LIN {X 0,Y 432.387,Z 300.627,A -85,B 0,C 180,E1 -9511.877,E2 -9511.877} C_VEL
LIN {X 0,Y 432.357,Z 300.63,A -85,B 0,C 180,E1 -9514.999,E2 -9514.999} C_VEL
LIN {X 0,Y 432.363,Z 300.629,A -85,B 0,C 180,E1 -9518.046,E2 -9518.046} C_VEL
LIN {X 0,Y 432.389,Z 300.628,A -85,B 0,C 180,E1 -9521.03,E2 -9521.03} C_VEL
LIN {X 0,Y 432.435,Z 300.621,A -85,B 0,C 180,E1 -9523.961,E2 -9523.961} C_VEL
LIN {X 0,Y 432.464,Z 300.618,A -85,B 0,C 180,E1 -9527.803,E2 -9527.803} C_VEL
LIN {X 0,Y 432.468,Z 300.616,A -85,B 0,C 180,E1 -9531.59,E2 -9531.59} C_VEL
LIN {X 0,Y 432.589,Z 300.602,A -85,B 0,C 180,E1 -9534.406,E2 -9534.406} C_VEL
LIN {X 0,Y 432.609,Z 300.601,A -85,B 0,C 180,E1 -9538.138,E2 -9538.138} C_VEL
LIN {X 0,Y 432.738,Z 300.585,A -85,B 0,C 180,E1 -9540,E2 -9540} C_VEL
LIN {X 0,Y 432.61,Z 300.6,A -85,B 0,C 180,E1 -9542.793,E2 -9542.793} C_VEL
LIN {X 0,Y 432.591,Z 300.602,A -85,B 0,C 180,E1 -9545.594,E2 -9545.594} C_VEL
LIN {X 0,Y 432.402,Z 300.627,A -85,B 0,C 180,E1 -9548.411,E2 -9548.411} C_VEL
LIN {X 0,Y 432.14,Z 300.66,A -85,B 0,C 180,E1 -9551.254,E2 -9551.254} C_VEL
LIN {X 0,Y 432.095,Z 301.406,A -85,B 0,C 180,E1 -9552.603,E2 -9552.603} C_VEL
LIN {X 0,Y 431.936,Z 304.726,A -85,B 0,C 180,E1 -9556.261,E2 -9556.261} C_VEL
LIN {X 0,Y 431.82,Z 307.511,A -85,B 0,C 180,E1 -9559.27,E2 -9559.27} C_VEL
LIN {X 0,Y 431.762,Z 309.431,A -85,B 0,C 180,E1 -9561.328,E2 -9561.328} C_VEL
LIN {X 0,Y 435.503,Z 322.776,A -85,B 0,C 180,E1 -9561.966,E2 -9561.966} C_VEL
LIN {X 0,Y 436.389,Z 326.305,A -85,B 0,C 180,E1 -9562.164,E2 -9562.164} C_VEL
LIN {X 0,Y 435.979,Z 338.712,A -85,B 0,C 180,E1 -9562.835,E2 -9562.835} C_VEL
LIN {X 0,Y 435.399,Z 349.849,A -85,B 0,C 180,E1 -9563.617,E2 -9563.617} C_VEL
LIN {X 0,Y 434.738,Z 360.847,A -85,B 0,C 180,E1 -9564.6,E2 -9564.6} C_VEL
LIN {X 0,Y 434.086,Z 370.626,A -85,B 0,C 180,E1 -9565.684,E2 -9565.684} C_VEL
LIN {X 0,Y 433.472,Z 380.219,A -85,B 0,C 180,E1 -9566.999,E2 -9566.999} C_VEL
LIN {X 0,Y 432.946,Z 388.349,A -85,B 0,C 180,E1 -9568.399,E2 -9568.399} C_VEL
LIN {X 0,Y 432.377,Z 395.707,A -85,B 0,C 180,E1 -9569.988,E2 -9569.988} C_VEL
LIN {X 0,Y 432.025,Z 400.707,A -85,B 0,C 180,E1 -9571.37,E2 -9571.37} C_VEL
LIN {X 0,Y 431.705,Z 405.281,A -85,B 0,C 180,E1 -9573.05,E2 -9573.05} C_VEL
LIN {X 0,Y 431.474,Z 408.451,A -85,B 0,C 180,E1 -9574.757,E2 -9574.757} C_VEL
LIN {X 0,Y 431.35,Z 409.815,A -85,B 0,C 180,E1 -9575.912,E2 -9575.912} C_VEL
LIN {X 0,Y 431.313,Z 410.554,A -85,B 0,C 180,E1 -9577.077,E2 -9577.077} C_VEL
LIN {X 0,Y 431.327,Z 410.608,A -85,B 0,C 180,E1 -9578.545,E2 -9578.545} C_VEL
LIN {X 0,Y 431.358,Z 409.677,A -85,B 0,C 180,E1 -9580.025,E2 -9580.025} C_VEL
LIN {X 0,Y 431.514,Z 407.052,A -85,B 0,C 180,E1 -9581.894,E2 -9581.894} C_VEL
LIN {X 0,Y 431.726,Z 404.385,A -85,B 0,C 180,E1 -9583.134,E2 -9583.134} C_VEL
LIN {X 0,Y 431.934,Z 399.792,A -85,B 0,C 180,E1 -9584.711,E2 -9584.711} C_VEL
LIN {X 0,Y 432.265,Z 393.586,A -85,B 0,C 180,E1 -9586.321,E2 -9586.321} C_VEL
LIN {X 0,Y 432.659,Z 387.205,A -85,B 0,C 180,E1 -9587.634,E2 -9587.634} C_VEL
LIN {X 0,Y 433.152,Z 379.47,A -85,B 0,C 180,E1 -9588.935,E2 -9588.935} C_VEL
LIN {X 0,Y 433.742,Z 370.118,A -85,B 0,C 180,E1 -9590.206,E2 -9590.206} C_VEL
LIN {X 0,Y 434.397,Z 359.637,A -85,B 0,C 180,E1 -9591.355,E2 -9591.355} C_VEL
LIN {X 0,Y 434.982,Z 348.401,A -85,B 0,C 180,E1 -9592.344,E2 -9592.344} C_VEL
LIN {X 0,Y 435.648,Z 335.625,A -85,B 0,C 180,E1 -9593.208,E2 -9593.208} C_VEL
LIN {X 0,Y 436.028,Z 326.289,A -85,B 0,C 180,E1 -9593.698,E2 -9593.698} C_VEL
LIN {X 0,Y 433.008,Z 313.174,A -85,B 0,C 180,E1 -9594.338,E2 -9594.338} C_VEL
LIN {X 0,Y 431.53,Z 307.479,A -85,B 0,C 180,E1 -9594.566,E2 -9594.566} C_VEL
LIN {X 0,Y 431.544,Z 304,A -85,B 0,C 180,E1 -9597.871,E2 -9597.871} C_VEL
LIN {X 0,Y 431.624,Z 301.006,A -85,B 0,C 180,E1 -9600.759,E2 -9600.759} C_VEL
LIN {X 0,Y 431.866,Z 300.693,A -85,B 0,C 180,E1 -9602.892,E2 -9602.892} C_VEL
LIN {X 0,Y 432.2,Z 300.649,A -85,B 0,C 180,E1 -9606.013,E2 -9606.013} C_VEL
LIN {X 0,Y 432.35,Z 300.631,A -85,B 0,C 180,E1 -9609.046,E2 -9609.046} C_VEL
LIN {X 0,Y 432.361,Z 300.628,A -85,B 0,C 180,E1 -9612.01,E2 -9612.01} C_VEL
LIN {X 0,Y 432.397,Z 300.627,A -85,B 0,C 180,E1 -9614.926,E2 -9614.926} C_VEL
LIN {X 0,Y 432.46,Z 300.615,A -85,B 0,C 180,E1 -9617.803,E2 -9617.803} C_VEL
LIN {X 0,Y 432.484,Z 300.612,A -85,B 0,C 180,E1 -9621.59,E2 -9621.59} C_VEL
LIN {X 0,Y 432.505,Z 300.61,A -85,B 0,C 180,E1 -9622.676,E2 -9622.676} C_VEL
LIN {X 0,Y 431.81,Z 300.698,A -85,B 0,C 180,E1 -9623.454,E2 -9623.454} C_VEL
LIN {X 0,Y 428.855,Z 301.067,A -85,B 0,C 180,E1 -9624.715,E2 -9624.715} C_VEL
LIN {X 0,Y 426.424,Z 301.367,A -85,B 0,C 180,E1 -9625.733,E2 -9625.733} C_VEL
LIN {X 0,Y 425.475,Z 301.487,A -85,B 0,C 180,E1 -9626.521,E2 -9626.521} C_VEL
LIN {X 0,Y 425.449,Z 301.488,A -85,B 0,C 180,E1 -9626.788,E2 -9626.788} C_VEL
LIN {X 0,Y 425.703,Z 301.457,A -85,B 0,C 180,E1 -9630,E2 -9630} C_VEL
LIN {X 0,Y 425.558,Z 301.478,A -85,B 0,C 180,E1 -9632.84,E2 -9632.84} C_VEL
LIN {X 0,Y 425.541,Z 301.477,A -85,B 0,C 180,E1 -9635.687,E2 -9635.687} C_VEL
LIN {X 0,Y 425.437,Z 301.494,A -85,B 0,C 180,E1 -9638.55,E2 -9638.55} C_VEL
LIN {X 0,Y 425.413,Z 301.497,A -85,B 0,C 180,E1 -9642.402,E2 -9642.402} C_VEL
LIN {X 0,Y 425.389,Z 301.5,A -85,B 0,C 180,E1 -9646.312,E2 -9646.312} C_VEL
LIN {X 0,Y 425.329,Z 301.504,A -85,B 0,C 180,E1 -9649.636,E2 -9649.636} C_VEL
LIN {X 0,Y 425.309,Z 301.506,A -85,B 0,C 180,E1 -9653.365,E2 -9653.365} C_VEL
LIN {X 0,Y 425.349,Z 301.502,A -85,B 0,C 180,E1 -9656.844,E2 -9656.844} C_VEL
LIN {X 0,Y 425.292,Z 301.511,A -85,B 0,C 180,E1 -9659.72,E2 -9659.72} C_VEL
LIN {X 0,Y 425.283,Z 301.509,A -85,B 0,C 180,E1 -9663.048,E2 -9663.048} C_VEL
LIN {X 0,Y 425.283,Z 301.513,A -85,B 0,C 180,E1 -9665.929,E2 -9665.929} C_VEL
LIN {X 0,Y 425.295,Z 301.508,A -85,B 0,C 180,E1 -9669.043,E2 -9669.043} C_VEL
LIN {X 0,Y 425.276,Z 301.51,A -85,B 0,C 180,E1 -9672.653,E2 -9672.653} C_VEL
LIN {X 0,Y 425.264,Z 301.514,A -85,B 0,C 180,E1 -9676.044,E2 -9676.044} C_VEL
LIN {X 0,Y 425.277,Z 301.51,A -85,B 0,C 180,E1 -9678.622,E2 -9678.622} C_VEL
LIN {X 0,Y 425.315,Z 301.506,A -85,B 0,C 180,E1 -9681.103,E2 -9681.103} C_VEL
LIN {X 0,Y 425.301,Z 301.507,A -85,B 0,C 180,E1 -9684.664,E2 -9684.664} C_VEL
LIN {X 0,Y 425.268,Z 301.513,A -85,B 0,C 180,E1 -9688.073,E2 -9688.073} C_VEL
LIN {X 0,Y 425.334,Z 301.506,A -85,B 0,C 180,E1 -9691.368,E2 -9691.368} C_VEL
LIN {X 0,Y 425.286,Z 301.509,A -85,B 0,C 180,E1 -9694.554,E2 -9694.554} C_VEL
LIN {X 0,Y 425.287,Z 301.509,A -85,B 0,C 180,E1 -9696.634,E2 -9696.634} C_VEL
LIN {X 0,Y 425.299,Z 301.51,A -85,B 0,C 180,E1 -9699.695,E2 -9699.695} C_VEL
LIN {X 0,Y 425.337,Z 301.503,A -85,B 0,C 180,E1 -9702.697,E2 -9702.697} C_VEL
LIN {X 0,Y 425.352,Z 301.501,A -85,B 0,C 180,E1 -9705.65,E2 -9705.65} C_VEL
LIN {X 0,Y 425.355,Z 301.502,A -85,B 0,C 180,E1 -9708.564,E2 -9708.564} C_VEL
LIN {X 0,Y 425.51,Z 301.482,A -85,B 0,C 180,E1 -9712.311,E2 -9712.311} C_VEL
LIN {X 0,Y 425.556,Z 301.475,A -85,B 0,C 180,E1 -9714.313,E2 -9714.313} C_VEL
LIN {X 0,Y 425.577,Z 301.472,A -85,B 0,C 180,E1 -9718.107,E2 -9718.107} C_VEL
LIN {X 0,Y 425.704,Z 301.457,A -85,B 0,C 180,E1 -9720,E2 -9720} C_VEL
LIN {X 0,Y 425.538,Z 301.48,A -85,B 0,C 180,E1 -9722.84,E2 -9722.84} C_VEL
LIN {X 0,Y 425.544,Z 301.476,A -85,B 0,C 180,E1 -9725.687,E2 -9725.687} C_VEL
LIN {X 0,Y 425.413,Z 301.495,A -85,B 0,C 180,E1 -9728.551,E2 -9728.551} C_VEL
LIN {X 0,Y 425.417,Z 301.495,A -85,B 0,C 180,E1 -9732.402,E2 -9732.402} C_VEL
LIN {X 0,Y 425.392,Z 301.498,A -85,B 0,C 180,E1 -9736.312,E2 -9736.312} C_VEL
LIN {X 0,Y 425.333,Z 301.504,A -85,B 0,C 180,E1 -9739.635,E2 -9739.635} C_VEL
LIN {X 0,Y 425.292,Z 301.512,A -85,B 0,C 180,E1 -9742.339,E2 -9742.339} C_VEL
LIN {X 0,Y 425.324,Z 301.507,A -85,B 0,C 180,E1 -9744.657,E2 -9744.657} C_VEL
LIN {X 0,Y 425.304,Z 301.508,A -85,B 0,C 180,E1 -9747.561,E2 -9747.561} C_VEL
LIN {X 0,Y 425.291,Z 301.51,A -85,B 0,C 180,E1 -9750.816,E2 -9750.816} C_VEL
LIN {X 0,Y 425.315,Z 301.508,A -85,B 0,C 180,E1 -9754.288,E2 -9754.288} C_VEL
LIN {X 0,Y 425.281,Z 301.511,A -85,B 0,C 180,E1 -9757.694,E2 -9757.694} C_VEL
LIN {X 0,Y 425.28,Z 301.513,A -85,B 0,C 180,E1 -9760.52,E2 -9760.52} C_VEL
LIN {X 0,Y 425.264,Z 301.514,A -85,B 0,C 180,E1 -9763.956,E2 -9763.956} C_VEL
LIN {X 0,Y 425.283,Z 301.51,A -85,B 0,C 180,E1 -9767.347,E2 -9767.347} C_VEL
LIN {X 0,Y 425.319,Z 301.554,A -85,B 0,C 180,E1 -9768.038,E2 -9768.038} C_VEL
LIN {X 0,Y 426.612,Z 308.704,A -85,B 0,C 180,E1 -9771.243,E2 -9771.243} C_VEL
LIN {X 0,Y 427.484,Z 314.493,A -85,B 0,C 180,E1 -9773.711,E2 -9773.711} C_VEL
LIN {X 0,Y 427.151,Z 320.214,A -85,B 0,C 180,E1 -9775.985,E2 -9775.985} C_VEL
LIN {X 0,Y 426.493,Z 328.818,A -85,B 0,C 180,E1 -9779.28,E2 -9779.28} C_VEL
LIN {X 0,Y 426.007,Z 335.947,A -85,B 0,C 180,E1 -9781.954,E2 -9781.954} C_VEL
LIN {X 0,Y 425.45,Z 345.144,A -85,B 0,C 180,E1 -9785.306,E2 -9785.306} C_VEL
LIN {X 0,Y 425.012,Z 354.577,A -85,B 0,C 180,E1 -9788.667,E2 -9788.667} C_VEL
LIN {X 0,Y 424.673,Z 364.594,A -85,B 0,C 180,E1 -9792.172,E2 -9792.172} C_VEL
LIN {X 0,Y 424.645,Z 367.488,A -85,B 0,C 180,E1 -9793.132,E2 -9793.132} C_VEL
LIN {X 0,Y 426.535,Z 381.53,A -85,B 0,C 180,E1 -9793.616,E2 -9793.616} C_VEL
LIN {X 0,Y 427.923,Z 394.874,A -85,B 0,C 180,E1 -9794.277,E2 -9794.277} C_VEL
LIN {X 0,Y 427.794,Z 403.089,A -85,B 0,C 180,E1 -9794.76,E2 -9794.76} C_VEL
LIN {X 0,Y 427.046,Z 414.476,A -85,B 0,C 180,E1 -9795.587,E2 -9795.587} C_VEL
LIN {X 0,Y 426.293,Z 426.083,A -85,B 0,C 180,E1 -9796.655,E2 -9796.655} C_VEL
LIN {X 0,Y 425.681,Z 436.413,A -85,B 0,C 180,E1 -9797.848,E2 -9797.848} C_VEL
LIN {X 0,Y 425.192,Z 444.822,A -85,B 0,C 180,E1 -9799.042,E2 -9799.042} C_VEL
LIN {X 0,Y 424.739,Z 453.057,A -85,B 0,C 180,E1 -9800.476,E2 -9800.476} C_VEL
LIN {X 0,Y 424.495,Z 459.692,A -85,B 0,C 180,E1 -9801.91,E2 -9801.91} C_VEL
LIN {X 0,Y 424.303,Z 464.964,A -85,B 0,C 180,E1 -9803.342,E2 -9803.342} C_VEL
LIN {X 0,Y 424.305,Z 469.053,A -85,B 0,C 180,E1 -9804.773,E2 -9804.773} C_VEL
LIN {X 0,Y 424.228,Z 472.054,A -85,B 0,C 180,E1 -9806.2,E2 -9806.2} C_VEL
LIN {X 0,Y 424.303,Z 473.512,A -85,B 0,C 180,E1 -9807.152,E2 -9807.152} C_VEL
LIN {X 0,Y 424.331,Z 474.525,A -85,B 0,C 180,E1 -9808.102,E2 -9808.102} C_VEL
LIN {X 0,Y 424.237,Z 475.342,A -85,B 0,C 180,E1 -9810,E2 -9810} C_VEL
LIN {X 0,Y 424.262,Z 475.126,A -85,B 0,C 180,E1 -9810.949,E2 -9810.949} C_VEL
LIN {X 0,Y 424.305,Z 474.488,A -85,B 0,C 180,E1 -9811.898,E2 -9811.898} C_VEL
LIN {X 0,Y 424.315,Z 473.449,A -85,B 0,C 180,E1 -9812.848,E2 -9812.848} C_VEL
LIN {X 0,Y 424.236,Z 471.996,A -85,B 0,C 180,E1 -9813.8,E2 -9813.8} C_VEL
LIN {X 0,Y 424.276,Z 468.966,A -85,B 0,C 180,E1 -9815.227,E2 -9815.227} C_VEL
LIN {X 0,Y 424.303,Z 464.877,A -85,B 0,C 180,E1 -9816.658,E2 -9816.658} C_VEL
LIN {X 0,Y 424.51,Z 458.627,A -85,B 0,C 180,E1 -9818.329,E2 -9818.329} C_VEL
LIN {X 0,Y 424.806,Z 451.808,A -85,B 0,C 180,E1 -9819.763,E2 -9819.763} C_VEL
LIN {X 0,Y 425.296,Z 443.38,A -85,B 0,C 180,E1 -9821.196,E2 -9821.196} C_VEL
LIN {X 0,Y 425.784,Z 434.788,A -85,B 0,C 180,E1 -9822.391,E2 -9822.391} C_VEL
LIN {X 0,Y 426.453,Z 424.473,A -85,B 0,C 180,E1 -9823.558,E2 -9823.558} C_VEL
LIN {X 0,Y 427.19,Z 413.873,A -85,B 0,C 180,E1 -9824.53,E2 -9824.53} C_VEL
LIN {X 0,Y 427.977,Z 402.662,A -85,B 0,C 180,E1 -9825.355,E2 -9825.355} C_VEL
LIN {X 0,Y 428.159,Z 395.858,A -85,B 0,C 180,E1 -9825.775,E2 -9825.775} C_VEL
LIN {X 0,Y 427.044,Z 382.25,A -85,B 0,C 180,E1 -9826.489,E2 -9826.489} C_VEL
LIN {X 0,Y 425.102,Z 368.516,A -85,B 0,C 180,E1 -9827.035,E2 -9827.035} C_VEL
LIN {X 0,Y 424.574,Z 365.324,A -85,B 0,C 180,E1 -9827.166,E2 -9827.166} C_VEL
LIN {X 0,Y 424.842,Z 356.134,A -85,B 0,C 180,E1 -9830.328,E2 -9830.328} C_VEL
LIN {X 0,Y 425.16,Z 347.485,A -85,B 0,C 180,E1 -9833.374,E2 -9833.374} C_VEL
LIN {X 0,Y 425.667,Z 337.704,A -85,B 0,C 180,E1 -9836.928,E2 -9836.928} C_VEL
LIN {X 0,Y 426.196,Z 329.072,A -85,B 0,C 180,E1 -9840.195,E2 -9840.195} C_VEL
LIN {X 0,Y 426.81,Z 322.215,A -85,B 0,C 180,E1 -9842.915,E2 -9842.915} C_VEL
LIN {X 0,Y 427.44,Z 315.509,A -85,B 0,C 180,E1 -9845.711,E2 -9845.711} C_VEL
LIN {X 0,Y 427.029,Z 310.899,A -85,B 0,C 180,E1 -9847.816,E2 -9847.816} C_VEL
LIN {X 0,Y 426.012,Z 305.245,A -85,B 0,C 180,E1 -9850.635,E2 -9850.635} C_VEL
LIN {X 0,Y 425.293,Z 301.513,A -85,B 0,C 180,E1 -9852.722,E2 -9852.722} C_VEL
LIN {X 0,Y 425.265,Z 301.519,A -85,B 0,C 180,E1 -9856.044,E2 -9856.044} C_VEL
LIN {X 0,Y 425.278,Z 301.515,A -85,B 0,C 180,E1 -9858.622,E2 -9858.622} C_VEL
LIN {X 0,Y 425.314,Z 301.511,A -85,B 0,C 180,E1 -9861.103,E2 -9861.103} C_VEL
LIN {X 0,Y 425.303,Z 301.51,A -85,B 0,C 180,E1 -9864.664,E2 -9864.664} C_VEL
LIN {X 0,Y 425.27,Z 301.515,A -85,B 0,C 180,E1 -9868.073,E2 -9868.073} C_VEL
LIN {X 0,Y 425.336,Z 301.505,A -85,B 0,C 180,E1 -9871.368,E2 -9871.368} C_VEL
LIN {X 0,Y 425.3,Z 301.509,A -85,B 0,C 180,E1 -9874.555,E2 -9874.555} C_VEL
LIN {X 0,Y 425.293,Z 301.508,A -85,B 0,C 180,E1 -9877.661,E2 -9877.661} C_VEL
LIN {X 0,Y 425.366,Z 301.501,A -85,B 0,C 180,E1 -9880.704,E2 -9880.704} C_VEL
LIN {X 0,Y 425.393,Z 301.498,A -85,B 0,C 180,E1 -9883.688,E2 -9883.688} C_VEL
LIN {X 0,Y 425.417,Z 301.495,A -85,B 0,C 180,E1 -9887.598,E2 -9887.598} C_VEL
LIN {X 0,Y 425.413,Z 301.494,A -85,B 0,C 180,E1 -9891.449,E2 -9891.449} C_VEL
LIN {X 0,Y 425.544,Z 301.48,A -85,B 0,C 180,E1 -9894.313,E2 -9894.313} C_VEL
LIN {X 0,Y 425.578,Z 301.476,A -85,B 0,C 180,E1 -9898.107,E2 -9898.107} C_VEL
LIN {X 0,Y 425.707,Z 301.46,A -85,B 0,C 180,E1 -9900,E2 -9900} C_VEL
LIN {X 0,Y 425.562,Z 301.478,A -85,B 0,C 180,E1 -9902.84,E2 -9902.84} C_VEL
LIN {X 0,Y 425.502,Z 301.484,A -85,B 0,C 180,E1 -9906.531,E2 -9906.531} C_VEL
LIN {X 0,Y 425.355,Z 301.505,A -85,B 0,C 180,E1 -9908.552,E2 -9908.552} C_VEL
LIN {X 0,Y 425.095,Z 301.538,A -85,B 0,C 180,E1 -9911.443,E2 -9911.443} C_VEL
LIN {X 0,Y 424.994,Z 303.079,A -85,B 0,C 180,E1 -9913.386,E2 -9913.386} C_VEL
LIN {X 0,Y 424.899,Z 305.791,A -85,B 0,C 180,E1 -9916.392,E2 -9916.392} C_VEL
LIN {X 0,Y 424.773,Z 308.564,A -85,B 0,C 180,E1 -9919.423,E2 -9919.423} C_VEL
LIN {X 0,Y 424.742,Z 310.014,A -85,B 0,C 180,E1 -9920.998,E2 -9920.998} C_VEL
LIN {X 0,Y 428.831,Z 324.498,A -85,B 0,C 180,E1 -9921.733,E2 -9921.733} C_VEL
LIN {X 0,Y 429.625,Z 328.745,A -85,B 0,C 180,E1 -9921.975,E2 -9921.975} C_VEL
LIN {X 0,Y 429.162,Z 340.386,A -85,B 0,C 180,E1 -9922.634,E2 -9922.634} C_VEL
LIN {X 0,Y 428.53,Z 351.475,A -85,B 0,C 180,E1 -9923.446,E2 -9923.446} C_VEL
LIN {X 0,Y 427.894,Z 361.547,A -85,B 0,C 180,E1 -9924.373,E2 -9924.373} C_VEL
LIN {X 0,Y 427.162,Z 372.189,A -85,B 0,C 180,E1 -9925.587,E2 -9925.587} C_VEL
LIN {X 0,Y 426.562,Z 380.521,A -85,B 0,C 180,E1 -9926.76,E2 -9926.76} C_VEL
LIN {X 0,Y 426.03,Z 388.001,A -85,B 0,C 180,E1 -9928.044,E2 -9928.044} C_VEL
LIN {X 0,Y 425.546,Z 393.963,A -85,B 0,C 180,E1 -9929.283,E2 -9929.283} C_VEL
LIN {X 0,Y 425.11,Z 399.897,A -85,B 0,C 180,E1 -9930.83,E2 -9930.83} C_VEL
LIN {X 0,Y 424.775,Z 404.653,A -85,B 0,C 180,E1 -9932.455,E2 -9932.455} C_VEL
LIN {X 0,Y 424.471,Z 408.375,A -85,B 0,C 180,E1 -9934.259,E2 -9934.259} C_VEL
LIN {X 0,Y 424.298,Z 410.269,A -85,B 0,C 180,E1 -9935.744,E2 -9935.744} C_VEL
LIN {X 0,Y 424.224,Z 411.191,A -85,B 0,C 180,E1 -9937.325,E2 -9937.325} C_VEL
LIN {X 0,Y 424.255,Z 410.955,A -85,B 0,C 180,E1 -9939.012,E2 -9939.012} C_VEL
LIN {X 0,Y 424.285,Z 409.891,A -85,B 0,C 180,E1 -9940.362,E2 -9940.362} C_VEL
LIN {X 0,Y 424.446,Z 407.785,A -85,B 0,C 180,E1 -9941.831,E2 -9941.831} C_VEL
LIN {X 0,Y 424.719,Z 403.846,A -85,B 0,C 180,E1 -9943.606,E2 -9943.606} C_VEL
LIN {X 0,Y 425.018,Z 398.531,A -85,B 0,C 180,E1 -9945.319,E2 -9945.319} C_VEL
LIN {X 0,Y 425.289,Z 393.211,A -85,B 0,C 180,E1 -9946.645,E2 -9946.645} C_VEL
LIN {X 0,Y 425.821,Z 385.574,A -85,B 0,C 180,E1 -9948.161,E2 -9948.161} C_VEL
LIN {X 0,Y 426.374,Z 377.198,A -85,B 0,C 180,E1 -9949.501,E2 -9949.501} C_VEL
LIN {X 0,Y 427.03,Z 367.293,A -85,B 0,C 180,E1 -9950.784,E2 -9950.784} C_VEL
LIN {X 0,Y 427.732,Z 356.075,A -85,B 0,C 180,E1 -9951.938,E2 -9951.938} C_VEL
LIN {X 0,Y 428.27,Z 345.278,A -85,B 0,C 180,E1 -9952.829,E2 -9952.829} C_VEL
LIN {X 0,Y 428.909,Z 332.666,A -85,B 0,C 180,E1 -9953.632,E2 -9953.632} C_VEL
LIN {X 0,Y 429.038,Z 326.59,A -85,B 0,C 180,E1 -9953.946,E2 -9953.946} C_VEL
LIN {X 0,Y 425.902,Z 313.545,A -85,B 0,C 180,E1 -9954.599,E2 -9954.599} C_VEL
LIN {X 0,Y 424.464,Z 307.924,A -85,B 0,C 180,E1 -9954.838,E2 -9954.838} C_VEL
LIN {X 0,Y 424.492,Z 304.616,A -85,B 0,C 180,E1 -9958.008,E2 -9958.008} C_VEL
LIN {X 0,Y 424.547,Z 302.32,A -85,B 0,C 180,E1 -9960.223,E2 -9960.223} C_VEL
LIN {X 0,Y 424.634,Z 301.597,A -85,B 0,C 180,E1 -9961.316,E2 -9961.316} C_VEL
LIN {X 0,Y 424.996,Z 301.546,A -85,B 0,C 180,E1 -9964.535,E2 -9964.535} C_VEL
LIN {X 0,Y 425.285,Z 301.511,A -85,B 0,C 180,E1 -9967.732,E2 -9967.732} C_VEL
LIN {X 0,Y 425.362,Z 301.5,A -85,B 0,C 180,E1 -9970.704,E2 -9970.704} C_VEL
LIN {X 0,Y 425.389,Z 301.496,A -85,B 0,C 180,E1 -9973.688,E2 -9973.688} C_VEL
LIN {X 0,Y 425.413,Z 301.493,A -85,B 0,C 180,E1 -9977.598,E2 -9977.598} C_VEL
LIN {X 0,Y 425.437,Z 301.491,A -85,B 0,C 180,E1 -9981.45,E2 -9981.45} C_VEL
LIN {X 0,Y 425.542,Z 301.479,A -85,B 0,C 180,E1 -9984.313,E2 -9984.313} C_VEL
LIN {X 0,Y 425.449,Z 301.488,A -85,B 0,C 180,E1 -9986.788,E2 -9986.788} C_VEL
LIN {X 0,Y 424.919,Z 301.557,A -85,B 0,C 180,E1 -9987.578,E2 -9987.578} C_VEL
LIN {X 0,Y 422.107,Z 301.913,A -85,B 0,C 180,E1 -9988.863,E2 -9988.863} C_VEL
LIN {X 0,Y 419.643,Z 302.22,A -85,B 0,C 180,E1 -9989.901,E2 -9989.901} C_VEL
LIN {X 0,Y 418.577,Z 302.349,A -85,B 0,C 180,E1 -9990.703,E2 -9990.703} C_VEL
LIN {X 0,Y 418.492,Z 302.357,A -85,B 0,C 180,E1 -9990.975,E2 -9990.975} C_VEL
LIN {X 0,Y 418.512,Z 302.356,A -85,B 0,C 180,E1 -9992.888,E2 -9992.888} C_VEL
LIN {X 0,Y 418.499,Z 302.355,A -85,B 0,C 180,E1 -9995.783,E2 -9995.783} C_VEL
LIN {X 0,Y 418.397,Z 302.37,A -85,B 0,C 180,E1 -9998.695,E2 -9998.695} C_VEL
LIN {X 0,Y 418.315,Z 302.377,A -85,B 0,C 180,E1 -10001.631,E2 -10001.631} C_VEL
LIN {X 0,Y 418.302,Z 302.382,A -85,B 0,C 180,E1 -10004.597,E2 -10004.597} C_VEL
LIN {X 0,Y 418.286,Z 302.381,A -85,B 0,C 180,E1 -10007.604,E2 -10007.604} C_VEL
LIN {X 0,Y 418.251,Z 302.387,A -85,B 0,C 180,E1 -10010.663,E2 -10010.663} C_VEL
LIN {X 0,Y 418.29,Z 302.381,A -85,B 0,C 180,E1 -10013.781,E2 -10013.781} C_VEL
LIN {X 0,Y 418.311,Z 302.377,A -85,B 0,C 180,E1 -10017.071,E2 -10017.071} C_VEL
LIN {X 0,Y 418.246,Z 302.389,A -85,B 0,C 180,E1 -10020.272,E2 -10020.272} C_VEL
LIN {X 0,Y 418.249,Z 302.388,A -85,B 0,C 180,E1 -10023.677,E2 -10023.677} C_VEL
LIN {X 0,Y 418.242,Z 302.387,A -85,B 0,C 180,E1 -10027.224,E2 -10027.224} C_VEL
LIN {X 0,Y 418.25,Z 302.387,A -85,B 0,C 180,E1 -10029.682,E2 -10029.682} C_VEL
LIN {X 0,Y 418.231,Z 302.39,A -85,B 0,C 180,E1 -10032.321,E2 -10032.321} C_VEL
LIN {X 0,Y 418.237,Z 302.387,A -85,B 0,C 180,E1 -10035.109,E2 -10035.109} C_VEL
LIN {X 0,Y 418.242,Z 302.39,A -85,B 0,C 180,E1 -10037.767,E2 -10037.767} C_VEL
LIN {X 0,Y 418.261,Z 302.384,A -85,B 0,C 180,E1 -10040.619,E2 -10040.619} C_VEL
LIN {X 0,Y 418.245,Z 302.389,A -85,B 0,C 180,E1 -10043.976,E2 -10043.976} C_VEL
LIN {X 0,Y 418.26,Z 302.386,A -85,B 0,C 180,E1 -10047.156,E2 -10047.156} C_VEL
LIN {X 0,Y 418.272,Z 302.383,A -85,B 0,C 180,E1 -10050.896,E2 -10050.896} C_VEL
LIN {X 0,Y 418.264,Z 302.384,A -85,B 0,C 180,E1 -10054.096,E2 -10054.096} C_VEL
LIN {X 0,Y 418.235,Z 302.39,A -85,B 0,C 180,E1 -10057.264,E2 -10057.264} C_VEL
LIN {X 0,Y 418.287,Z 302.381,A -85,B 0,C 180,E1 -10060.364,E2 -10060.364} C_VEL
LIN {X 0,Y 418.321,Z 302.379,A -85,B 0,C 180,E1 -10063.405,E2 -10063.405} C_VEL
LIN {X 0,Y 418.351,Z 302.376,A -85,B 0,C 180,E1 -10066.999,E2 -10066.999} C_VEL
LIN {X 0,Y 418.343,Z 302.373,A -85,B 0,C 180,E1 -10070.329,E2 -10070.329} C_VEL
LIN {X 0,Y 418.484,Z 302.359,A -85,B 0,C 180,E1 -10073.249,E2 -10073.249} C_VEL
LIN {X 0,Y 418.34,Z 302.376,A -85,B 0,C 180,E1 -10075.182,E2 -10075.182} C_VEL
LIN {X 0,Y 418.546,Z 302.348,A -85,B 0,C 180,E1 -10078.076,E2 -10078.076} C_VEL
LIN {X 0,Y 418.674,Z 302.333,A -85,B 0,C 180,E1 -10080,E2 -10080} C_VEL
LIN {X 0,Y 418.493,Z 302.358,A -85,B 0,C 180,E1 -10082.888,E2 -10082.888} C_VEL
LIN {X 0,Y 418.502,Z 302.353,A -85,B 0,C 180,E1 -10085.783,E2 -10085.783} C_VEL
LIN {X 0,Y 418.382,Z 302.372,A -85,B 0,C 180,E1 -10088.696,E2 -10088.696} C_VEL
LIN {X 0,Y 418.32,Z 302.377,A -85,B 0,C 180,E1 -10091.631,E2 -10091.631} C_VEL
LIN {X 0,Y 418.306,Z 302.381,A -85,B 0,C 180,E1 -10094.597,E2 -10094.597} C_VEL
LIN {X 0,Y 418.284,Z 302.38,A -85,B 0,C 180,E1 -10097.604,E2 -10097.604} C_VEL
LIN {X 0,Y 418.254,Z 302.388,A -85,B 0,C 180,E1 -10100.663,E2 -10100.663} C_VEL
LIN {X 0,Y 418.279,Z 302.383,A -85,B 0,C 180,E1 -10103.782,E2 -10103.782} C_VEL
LIN {X 0,Y 418.27,Z 302.384,A -85,B 0,C 180,E1 -10107.059,E2 -10107.059} C_VEL
LIN {X 0,Y 418.246,Z 302.389,A -85,B 0,C 180,E1 -10110.272,E2 -10110.272} C_VEL
LIN {X 0,Y 418.252,Z 302.385,A -85,B 0,C 180,E1 -10113.677,E2 -10113.677} C_VEL
LIN {X 0,Y 418.243,Z 302.385,A -85,B 0,C 180,E1 -10117.224,E2 -10117.224} C_VEL
LIN {X 0,Y 418.245,Z 302.388,A -85,B 0,C 180,E1 -10119.683,E2 -10119.683} C_VEL
LIN {X 0,Y 418.227,Z 302.39,A -85,B 0,C 180,E1 -10122.32,E2 -10122.32} C_VEL
LIN {X 0,Y 418.239,Z 302.387,A -85,B 0,C 180,E1 -10125.109,E2 -10125.109} C_VEL
LIN {X 0,Y 418.273,Z 302.467,A -85,B 0,C 180,E1 -10127.77,E2 -10127.77} C_VEL
LIN {X 0,Y 419.585,Z 309.715,A -85,B 0,C 180,E1 -10131.088,E2 -10131.088} C_VEL
LIN {X 0,Y 420.443,Z 314.916,A -85,B 0,C 180,E1 -10133.356,E2 -10133.356} C_VEL
LIN {X 0,Y 420.247,Z 319.797,A -85,B 0,C 180,E1 -10135.347,E2 -10135.347} C_VEL
LIN {X 0,Y 419.657,Z 326.932,A -85,B 0,C 180,E1 -10138.161,E2 -10138.161} C_VEL
LIN {X 0,Y 419.068,Z 335.497,A -85,B 0,C 180,E1 -10141.447,E2 -10141.447} C_VEL
LIN {X 0,Y 418.428,Z 345.286,A -85,B 0,C 180,E1 -10145.094,E2 -10145.094} C_VEL
LIN {X 0,Y 417.978,Z 354.077,A -85,B 0,C 180,E1 -10148.289,E2 -10148.289} C_VEL
LIN {X 0,Y 417.617,Z 364.048,A -85,B 0,C 180,E1 -10151.86,E2 -10151.86} C_VEL
LIN {X 0,Y 417.56,Z 366.863,A -85,B 0,C 180,E1 -10152.857,E2 -10152.857} C_VEL
LIN {X 0,Y 419.506,Z 381.115,A -85,B 0,C 180,E1 -10153.363,E2 -10153.363} C_VEL
LIN {X 0,Y 420.824,Z 394.09,A -85,B 0,C 180,E1 -10154.016,E2 -10154.016} C_VEL
LIN {X 0,Y 420.999,Z 400.277,A -85,B 0,C 180,E1 -10154.387,E2 -10154.387} C_VEL
LIN {X 0,Y 420.262,Z 412.205,A -85,B 0,C 180,E1 -10155.225,E2 -10155.225} C_VEL
LIN {X 0,Y 419.502,Z 422.969,A -85,B 0,C 180,E1 -10156.188,E2 -10156.188} C_VEL
LIN {X 0,Y 418.812,Z 433.778,A -85,B 0,C 180,E1 -10157.399,E2 -10157.399} C_VEL
LIN {X 0,Y 418.276,Z 442.586,A -85,B 0,C 180,E1 -10158.613,E2 -10158.613} C_VEL
LIN {X 0,Y 417.732,Z 451.157,A -85,B 0,C 180,E1 -10160.07,E2 -10160.07} C_VEL
LIN {X 0,Y 417.452,Z 458.041,A -85,B 0,C 180,E1 -10161.529,E2 -10161.529} C_VEL
LIN {X 0,Y 417.234,Z 464.357,A -85,B 0,C 180,E1 -10163.228,E2 -10163.228} C_VEL
LIN {X 0,Y 417.211,Z 468.462,A -85,B 0,C 180,E1 -10164.684,E2 -10164.684} C_VEL
LIN {X 0,Y 417.138,Z 471.48,A -85,B 0,C 180,E1 -10166.136,E2 -10166.136} C_VEL
LIN {X 0,Y 417.231,Z 472.953,A -85,B 0,C 180,E1 -10167.103,E2 -10167.103} C_VEL
LIN {X 0,Y 417.247,Z 473.972,A -85,B 0,C 180,E1 -10168.069,E2 -10168.069} C_VEL
LIN {X 0,Y 417.206,Z 474.586,A -85,B 0,C 180,E1 -10169.035,E2 -10169.035} C_VEL
LIN {X 0,Y 417.179,Z 474.802,A -85,B 0,C 180,E1 -10170,E2 -10170} C_VEL
LIN {X 0,Y 417.206,Z 474.597,A -85,B 0,C 180,E1 -10170.965,E2 -10170.965} C_VEL
LIN {X 0,Y 417.224,Z 473.961,A -85,B 0,C 180,E1 -10171.931,E2 -10171.931} C_VEL
LIN {X 0,Y 417.241,Z 472.925,A -85,B 0,C 180,E1 -10172.897,E2 -10172.897} C_VEL
LIN {X 0,Y 417.143,Z 471.473,A -85,B 0,C 180,E1 -10173.864,E2 -10173.864} C_VEL
LIN {X 0,Y 417.185,Z 468.449,A -85,B 0,C 180,E1 -10175.316,E2 -10175.316} C_VEL
LIN {X 0,Y 417.234,Z 464.366,A -85,B 0,C 180,E1 -10176.772,E2 -10176.772} C_VEL
LIN {X 0,Y 417.448,Z 458.128,A -85,B 0,C 180,E1 -10178.471,E2 -10178.471} C_VEL
LIN {X 0,Y 417.763,Z 451.314,A -85,B 0,C 180,E1 -10179.93,E2 -10179.93} C_VEL
LIN {X 0,Y 418.296,Z 442.905,A -85,B 0,C 180,E1 -10181.386,E2 -10181.386} C_VEL
LIN {X 0,Y 418.812,Z 434.353,A -85,B 0,C 180,E1 -10182.601,E2 -10182.601} C_VEL
LIN {X 0,Y 419.507,Z 424.104,A -85,B 0,C 180,E1 -10183.787,E2 -10183.787} C_VEL
LIN {X 0,Y 420.325,Z 413.577,A -85,B 0,C 180,E1 -10184.773,E2 -10184.773} C_VEL
LIN {X 0,Y 421.099,Z 402.436,A -85,B 0,C 180,E1 -10185.612,E2 -10185.612} C_VEL
LIN {X 0,Y 421.201,Z 395.721,A -85,B 0,C 180,E1 -10186.043,E2 -10186.043} C_VEL
LIN {X 0,Y 420.068,Z 382.084,A -85,B 0,C 180,E1 -10186.781,E2 -10186.781} C_VEL
LIN {X 0,Y 418.199,Z 368.878,A -85,B 0,C 180,E1 -10187.328,E2 -10187.328} C_VEL
LIN {X 0,Y 417.495,Z 364.75,A -85,B 0,C 180,E1 -10187.488,E2 -10187.488} C_VEL
LIN {X 0,Y 417.828,Z 355.672,A -85,B 0,C 180,E1 -10190.685,E2 -10190.685} C_VEL
LIN {X 0,Y 418.124,Z 347.068,A -85,B 0,C 180,E1 -10193.791,E2 -10193.791} C_VEL
LIN {X 0,Y 418.646,Z 337.992,A -85,B 0,C 180,E1 -10197.16,E2 -10197.16} C_VEL
LIN {X 0,Y 419.302,Z 328.805,A -85,B 0,C 180,E1 -10200.737,E2 -10200.737} C_VEL
LIN {X 0,Y 419.908,Z 321.977,A -85,B 0,C 180,E1 -10203.527,E2 -10203.527} C_VEL
LIN {X 0,Y 420.474,Z 316.662,A -85,B 0,C 180,E1 -10205.804,E2 -10205.804} C_VEL
LIN {X 0,Y 420.157,Z 312.851,A -85,B 0,C 180,E1 -10207.569,E2 -10207.569} C_VEL
LIN {X 0,Y 418.992,Z 306.137,A -85,B 0,C 180,E1 -10210.991,E2 -10210.991} C_VEL
LIN {X 0,Y 418.243,Z 302.391,A -85,B 0,C 180,E1 -10213.149,E2 -10213.149} C_VEL
LIN {X 0,Y 418.213,Z 302.399,A -85,B 0,C 180,E1 -10216.449,E2 -10216.449} C_VEL
LIN {X 0,Y 418.227,Z 302.396,A -85,B 0,C 180,E1 -10219.13,E2 -10219.13} C_VEL
LIN {X 0,Y 418.233,Z 302.392,A -85,B 0,C 180,E1 -10222.167,E2 -10222.167} C_VEL
LIN {X 0,Y 418.269,Z 302.384,A -85,B 0,C 180,E1 -10225.42,E2 -10225.42} C_VEL
LIN {X 0,Y 418.216,Z 302.392,A -85,B 0,C 180,E1 -10228.604,E2 -10228.604} C_VEL
LIN {X 0,Y 418.297,Z 302.382,A -85,B 0,C 180,E1 -10231.937,E2 -10231.937} C_VEL
LIN {X 0,Y 418.294,Z 302.38,A -85,B 0,C 180,E1 -10235.163,E2 -10235.163} C_VEL
LIN {X 0,Y 418.239,Z 302.389,A -85,B 0,C 180,E1 -10238.304,E2 -10238.304} C_VEL
LIN {X 0,Y 418.286,Z 302.383,A -85,B 0,C 180,E1 -10241.383,E2 -10241.383} C_VEL
LIN {X 0,Y 418.307,Z 302.378,A -85,B 0,C 180,E1 -10244.406,E2 -10244.406} C_VEL
LIN {X 0,Y 418.361,Z 302.374,A -85,B 0,C 180,E1 -10247.386,E2 -10247.386} C_VEL
LIN {X 0,Y 418.344,Z 302.376,A -85,B 0,C 180,E1 -10250.329,E2 -10250.329} C_VEL
LIN {X 0,Y 418.463,Z 302.36,A -85,B 0,C 180,E1 -10253.248,E2 -10253.248} C_VEL
LIN {X 0,Y 418.338,Z 302.376,A -85,B 0,C 180,E1 -10255.181,E2 -10255.181} C_VEL
LIN {X 0,Y 418.547,Z 302.352,A -85,B 0,C 180,E1 -10258.075,E2 -10258.075} C_VEL
LIN {X 0,Y 418.676,Z 302.336,A -85,B 0,C 180,E1 -10260,E2 -10260} C_VEL
LIN {X 0,Y 418.515,Z 302.356,A -85,B 0,C 180,E1 -10262.888,E2 -10262.888} C_VEL
LIN {X 0,Y 418.463,Z 302.36,A -85,B 0,C 180,E1 -10266.53,E2 -10266.53} C_VEL
LIN {X 0,Y 418.304,Z 302.383,A -85,B 0,C 180,E1 -10268.697,E2 -10268.697} C_VEL
LIN {X 0,Y 418.06,Z 302.532,A -85,B 0,C 180,E1 -10271.638,E2 -10271.638} C_VEL
LIN {X 0,Y 417.92,Z 305.149,A -85,B 0,C 180,E1 -10274.611,E2 -10274.611} C_VEL
LIN {X 0,Y 417.773,Z 307.854,A -85,B 0,C 180,E1 -10277.626,E2 -10277.626} C_VEL
LIN {X 0,Y 417.718,Z 310.831,A -85,B 0,C 180,E1 -10280.69,E2 -10280.69} C_VEL
LIN {X 0,Y 421.663,Z 324.251,A -85,B 0,C 180,E1 -10281.383,E2 -10281.383} C_VEL
LIN {X 0,Y 422.882,Z 329.629,A -85,B 0,C 180,E1 -10281.702,E2 -10281.702} C_VEL
LIN {X 0,Y 422.41,Z 341.168,A -85,B 0,C 180,E1 -10282.37,E2 -10282.37} C_VEL
LIN {X 0,Y 421.748,Z 352.071,A -85,B 0,C 180,E1 -10283.184,E2 -10283.184} C_VEL
LIN {X 0,Y 421.045,Z 362.279,A -85,B 0,C 180,E1 -10284.139,E2 -10284.139} C_VEL
LIN {X 0,Y 420.299,Z 372.513,A -85,B 0,C 180,E1 -10285.325,E2 -10285.325} C_VEL
LIN {X 0,Y 419.616,Z 381.531,A -85,B 0,C 180,E1 -10286.617,E2 -10286.617} C_VEL
LIN {X 0,Y 419.02,Z 389.352,A -85,B 0,C 180,E1 -10288.01,E2 -10288.01} C_VEL
LIN {X 0,Y 418.481,Z 395.773,A -85,B 0,C 180,E1 -10289.421,E2 -10289.421} C_VEL
LIN {X 0,Y 418.032,Z 401.372,A -85,B 0,C 180,E1 -10290.971,E2 -10290.971} C_VEL
LIN {X 0,Y 417.668,Z 406.111,A -85,B 0,C 180,E1 -10292.718,E2 -10292.718} C_VEL
LIN {X 0,Y 417.372,Z 409.248,A -85,B 0,C 180,E1 -10294.401,E2 -10294.401} C_VEL
LIN {X 0,Y 417.204,Z 411.156,A -85,B 0,C 180,E1 -10296.128,E2 -10296.128} C_VEL
LIN {X 0,Y 417.162,Z 411.772,A -85,B 0,C 180,E1 -10297.644,E2 -10297.644} C_VEL
LIN {X 0,Y 417.194,Z 411.386,A -85,B 0,C 180,E1 -10299.202,E2 -10299.202} C_VEL
LIN {X 0,Y 417.256,Z 409.591,A -85,B 0,C 180,E1 -10301.063,E2 -10301.063} C_VEL
LIN {X 0,Y 417.569,Z 406.088,A -85,B 0,C 180,E1 -10302.972,E2 -10302.972} C_VEL
LIN {X 0,Y 417.815,Z 401.728,A -85,B 0,C 180,E1 -10304.609,E2 -10304.609} C_VEL
LIN {X 0,Y 418.14,Z 395.763,A -85,B 0,C 180,E1 -10306.281,E2 -10306.281} C_VEL
LIN {X 0,Y 418.6,Z 388.737,A -85,B 0,C 180,E1 -10307.811,E2 -10307.811} C_VEL
LIN {X 0,Y 419.143,Z 381.057,A -85,B 0,C 180,E1 -10309.161,E2 -10309.161} C_VEL
LIN {X 0,Y 419.81,Z 371.699,A -85,B 0,C 180,E1 -10310.494,E2 -10310.494} C_VEL
LIN {X 0,Y 420.527,Z 361.459,A -85,B 0,C 180,E1 -10311.666,E2 -10311.666} C_VEL
LIN {X 0,Y 421.107,Z 351.207,A -85,B 0,C 180,E1 -10312.621,E2 -10312.621} C_VEL
LIN {X 0,Y 421.732,Z 340.479,A -85,B 0,C 180,E1 -10313.422,E2 -10313.422} C_VEL
LIN {X 0,Y 422.253,Z 328.356,A -85,B 0,C 180,E1 -10314.122,E2 -10314.122} C_VEL
LIN {X 0,Y 419.169,Z 315.26,A -85,B 0,C 180,E1 -10314.805,E2 -10314.805} C_VEL
LIN {X 0,Y 417.432,Z 308.386,A -85,B 0,C 180,E1 -10315.117,E2 -10315.117} C_VEL
LIN {X 0,Y 417.442,Z 304.816,A -85,B 0,C 180,E1 -10318.539,E2 -10318.539} C_VEL
LIN {X 0,Y 417.51,Z 302.512,A -85,B 0,C 180,E1 -10320.78,E2 -10320.78} C_VEL
LIN {X 0,Y 417.904,Z 302.429,A -85,B 0,C 180,E1 -10324.071,E2 -10324.071} C_VEL
LIN {X 0,Y 418.197,Z 302.395,A -85,B 0,C 180,E1 -10327.261,E2 -10327.261} C_VEL
LIN {X 0,Y 418.284,Z 302.38,A -85,B 0,C 180,E1 -10330.364,E2 -10330.364} C_VEL
LIN {X 0,Y 418.317,Z 302.379,A -85,B 0,C 180,E1 -10333.404,E2 -10333.404} C_VEL
LIN {X 0,Y 418.348,Z 302.376,A -85,B 0,C 180,E1 -10336.999,E2 -10336.999} C_VEL
LIN {X 0,Y 418.341,Z 302.375,A -85,B 0,C 180,E1 -10340.329,E2 -10340.329} C_VEL
LIN {X 0,Y 418.46,Z 302.361,A -85,B 0,C 180,E1 -10343.248,E2 -10343.248} C_VEL
LIN {X 0,Y 418.337,Z 302.377,A -85,B 0,C 180,E1 -10345.181,E2 -10345.181} C_VEL
LIN {X 0,Y 418.543,Z 302.35,A -85,B 0,C 180,E1 -10348.075,E2 -10348.075} C_VEL
LIN {X 0,Y 418.672,Z 302.332,A -85,B 0,C 180,E1 -10350,E2 -10350} C_VEL
LIN {X 0,Y 418.492,Z 302.357,A -85,B 0,C 180,E1 -10350.975,E2 -10350.975} C_VEL
LIN {X 0,Y 417.803,Z 302.442,A -85,B 0,C 180,E1 -10351.778,E2 -10351.778} C_VEL
LIN {X 0,Y 414.857,Z 302.81,A -85,B 0,C 180,E1 -10353.08,E2 -10353.08} C_VEL
LIN {X 0,Y 412.399,Z 303.117,A -85,B 0,C 180,E1 -10354.131,E2 -10354.131} C_VEL
LIN {X 0,Y 411.394,Z 303.241,A -85,B 0,C 180,E1 -10354.946,E2 -10354.946} C_VEL
LIN {X 0,Y 411.339,Z 303.246,A -85,B 0,C 180,E1 -10355.221,E2 -10355.221} C_VEL
LIN {X 0,Y 411.389,Z 303.24,A -85,B 0,C 180,E1 -10357.855,E2 -10357.855} C_VEL
LIN {X 0,Y 411.286,Z 303.256,A -85,B 0,C 180,E1 -10360.834,E2 -10360.834} C_VEL
LIN {X 0,Y 411.255,Z 303.258,A -85,B 0,C 180,E1 -10363.842,E2 -10363.842} C_VEL
LIN {X 0,Y 411.258,Z 303.258,A -85,B 0,C 180,E1 -10366.889,E2 -10366.889} C_VEL
LIN {X 0,Y 411.232,Z 303.261,A -85,B 0,C 180,E1 -10369.987,E2 -10369.987} C_VEL
LIN {X 0,Y 411.205,Z 303.262,A -85,B 0,C 180,E1 -10373.148,E2 -10373.148} C_VEL
LIN {X 0,Y 411.239,Z 303.262,A -85,B 0,C 180,E1 -10376.381,E2 -10376.381} C_VEL
LIN {X 0,Y 411.202,Z 303.265,A -85,B 0,C 180,E1 -10379.713,E2 -10379.713} C_VEL
LIN {X 0,Y 411.208,Z 303.262,A -85,B 0,C 180,E1 -10383.156,E2 -10383.156} C_VEL
LIN {X 0,Y 411.194,Z 303.265,A -85,B 0,C 180,E1 -10386.553,E2 -10386.553} C_VEL
LIN {X 0,Y 411.214,Z 303.264,A -85,B 0,C 180,E1 -10389.728,E2 -10389.728} C_VEL
LIN {X 0,Y 411.175,Z 303.267,A -85,B 0,C 180,E1 -10393.134,E2 -10393.134} C_VEL
LIN {X 0,Y 411.17,Z 303.27,A -85,B 0,C 180,E1 -10395.881,E2 -10395.881} C_VEL
LIN {X 0,Y 411.167,Z 303.267,A -85,B 0,C 180,E1 -10398.772,E2 -10398.772} C_VEL
LIN {X 0,Y 411.21,Z 303.265,A -85,B 0,C 180,E1 -10401.831,E2 -10401.831} C_VEL
LIN {X 0,Y 411.212,Z 303.263,A -85,B 0,C 180,E1 -10405.122,E2 -10405.122} C_VEL
LIN {X 0,Y 411.168,Z 303.269,A -85,B 0,C 180,E1 -10408.003,E2 -10408.003} C_VEL
LIN {X 0,Y 411.221,Z 303.264,A -85,B 0,C 180,E1 -10411.41,E2 -10411.41} C_VEL
LIN {X 0,Y 411.236,Z 303.262,A -85,B 0,C 180,E1 -10413.619,E2 -10413.619} C_VEL
LIN {X 0,Y 411.199,Z 303.265,A -85,B 0,C 180,E1 -10416.852,E2 -10416.852} C_VEL
LIN {X 0,Y 411.219,Z 303.262,A -85,B 0,C 180,E1 -10420.051,E2 -10420.051} C_VEL
LIN {X 0,Y 411.267,Z 303.258,A -85,B 0,C 180,E1 -10423.131,E2 -10423.131} C_VEL
LIN {X 0,Y 411.31,Z 303.253,A -85,B 0,C 180,E1 -10426.896,E2 -10426.896} C_VEL
LIN {X 0,Y 411.296,Z 303.251,A -85,B 0,C 180,E1 -10430.161,E2 -10430.161} C_VEL
LIN {X 0,Y 411.447,Z 303.237,A -85,B 0,C 180,E1 -10433.133,E2 -10433.133} C_VEL
LIN {X 0,Y 411.312,Z 303.252,A -85,B 0,C 180,E1 -10435.099,E2 -10435.099} C_VEL
LIN {X 0,Y 411.514,Z 303.223,A -85,B 0,C 180,E1 -10438.043,E2 -10438.043} C_VEL
LIN {X 0,Y 411.643,Z 303.208,A -85,B 0,C 180,E1 -10440,E2 -10440} C_VEL
LIN {X 0,Y 411.45,Z 303.235,A -85,B 0,C 180,E1 -10442.937,E2 -10442.937} C_VEL
LIN {X 0,Y 411.427,Z 303.238,A -85,B 0,C 180,E1 -10446.868,E2 -10446.868} C_VEL
LIN {X 0,Y 411.296,Z 303.25,A -85,B 0,C 180,E1 -10449.839,E2 -10449.839} C_VEL
LIN {X 0,Y 411.31,Z 303.25,A -85,B 0,C 180,E1 -10453.104,E2 -10453.104} C_VEL
LIN {X 0,Y 411.261,Z 303.257,A -85,B 0,C 180,E1 -10456.889,E2 -10456.889} C_VEL
LIN {X 0,Y 411.235,Z 303.261,A -85,B 0,C 180,E1 -10459.987,E2 -10459.987} C_VEL
LIN {X 0,Y 411.2,Z 303.264,A -85,B 0,C 180,E1 -10463.148,E2 -10463.148} C_VEL
LIN {X 0,Y 411.207,Z 303.265,A -85,B 0,C 180,E1 -10466.383,E2 -10466.383} C_VEL
LIN {X 0,Y 411.202,Z 303.263,A -85,B 0,C 180,E1 -10469.713,E2 -10469.713} C_VEL
LIN {X 0,Y 411.21,Z 303.261,A -85,B 0,C 180,E1 -10473.156,E2 -10473.156} C_VEL
LIN {X 0,Y 411.196,Z 303.265,A -85,B 0,C 180,E1 -10476.552,E2 -10476.552} C_VEL
LIN {X 0,Y 411.21,Z 303.265,A -85,B 0,C 180,E1 -10479.727,E2 -10479.727} C_VEL
LIN {X 0,Y 411.174,Z 303.269,A -85,B 0,C 180,E1 -10483.134,E2 -10483.134} C_VEL
LIN {X 0,Y 411.17,Z 303.268,A -85,B 0,C 180,E1 -10485.881,E2 -10485.881} C_VEL
LIN {X 0,Y 411.233,Z 303.446,A -85,B 0,C 180,E1 -10487.531,E2 -10487.531} C_VEL
LIN {X 0,Y 412.58,Z 310.725,A -85,B 0,C 180,E1 -10490.93,E2 -10490.93} C_VEL
LIN {X 0,Y 413.482,Z 316.504,A -85,B 0,C 180,E1 -10493.494,E2 -10493.494} C_VEL
LIN {X 0,Y 413.153,Z 322.216,A -85,B 0,C 180,E1 -10495.85,E2 -10495.85} C_VEL
LIN {X 0,Y 412.432,Z 330.781,A -85,B 0,C 180,E1 -10499.255,E2 -10499.255} C_VEL
LIN {X 0,Y 411.821,Z 339.324,A -85,B 0,C 180,E1 -10502.563,E2 -10502.563} C_VEL
LIN {X 0,Y 411.227,Z 347.846,A -85,B 0,C 180,E1 -10505.784,E2 -10505.784} C_VEL
LIN {X 0,Y 410.773,Z 357.807,A -85,B 0,C 180,E1 -10509.467,E2 -10509.467} C_VEL
LIN {X 0,Y 410.473,Z 366.348,A -85,B 0,C 180,E1 -10512.565,E2 -10512.565} C_VEL
LIN {X 0,Y 412.528,Z 381.507,A -85,B 0,C 180,E1 -10513.136,E2 -10513.136} C_VEL
LIN {X 0,Y 413.818,Z 393.884,A -85,B 0,C 180,E1 -10513.782,E2 -10513.782} C_VEL
LIN {X 0,Y 414.093,Z 399.531,A -85,B 0,C 180,E1 -10514.131,E2 -10514.131} C_VEL
LIN {X 0,Y 413.331,Z 411.362,A -85,B 0,C 180,E1 -10514.971,E2 -10514.971} C_VEL
LIN {X 0,Y 412.53,Z 422.203,A -85,B 0,C 180,E1 -10515.95,E2 -10515.95} C_VEL
LIN {X 0,Y 411.859,Z 433.055,A -85,B 0,C 180,E1 -10517.183,E2 -10517.183} C_VEL
LIN {X 0,Y 411.273,Z 441.894,A -85,B 0,C 180,E1 -10518.417,E2 -10518.417} C_VEL
LIN {X 0,Y 410.677,Z 450.504,A -85,B 0,C 180,E1 -10519.897,E2 -10519.897} C_VEL
LIN {X 0,Y 410.375,Z 457.411,A -85,B 0,C 180,E1 -10521.382,E2 -10521.382} C_VEL
LIN {X 0,Y 410.166,Z 463.749,A -85,B 0,C 180,E1 -10523.111,E2 -10523.111} C_VEL
LIN {X 0,Y 410.121,Z 467.871,A -85,B 0,C 180,E1 -10524.592,E2 -10524.592} C_VEL
LIN {X 0,Y 410.05,Z 470.905,A -85,B 0,C 180,E1 -10526.069,E2 -10526.069} C_VEL
LIN {X 0,Y 410.16,Z 472.395,A -85,B 0,C 180,E1 -10527.053,E2 -10527.053} C_VEL
LIN {X 0,Y 410.167,Z 473.42,A -85,B 0,C 180,E1 -10528.036,E2 -10528.036} C_VEL
LIN {X 0,Y 410.152,Z 474.04,A -85,B 0,C 180,E1 -10529.018,E2 -10529.018} C_VEL
LIN {X 0,Y 410.123,Z 474.261,A -85,B 0,C 180,E1 -10530,E2 -10530} C_VEL
LIN {X 0,Y 410.151,Z 474.068,A -85,B 0,C 180,E1 -10530.982,E2 -10530.982} C_VEL
LIN {X 0,Y 410.146,Z 473.434,A -85,B 0,C 180,E1 -10531.964,E2 -10531.964} C_VEL
LIN {X 0,Y 410.169,Z 472.4,A -85,B 0,C 180,E1 -10532.947,E2 -10532.947} C_VEL
LIN {X 0,Y 410.052,Z 470.95,A -85,B 0,C 180,E1 -10533.931,E2 -10533.931} C_VEL
LIN {X 0,Y 410.098,Z 467.932,A -85,B 0,C 180,E1 -10535.409,E2 -10535.409} C_VEL
LIN {X 0,Y 410.165,Z 463.859,A -85,B 0,C 180,E1 -10536.889,E2 -10536.889} C_VEL
LIN {X 0,Y 410.37,Z 457.645,A -85,B 0,C 180,E1 -10538.618,E2 -10538.618} C_VEL
LIN {X 0,Y 410.699,Z 450.859,A -85,B 0,C 180,E1 -10540.102,E2 -10540.102} C_VEL
LIN {X 0,Y 411.279,Z 442.48,A -85,B 0,C 180,E1 -10541.583,E2 -10541.583} C_VEL
LIN {X 0,Y 411.861,Z 433.956,A -85,B 0,C 180,E1 -10542.817,E2 -10542.817} C_VEL
LIN {X 0,Y 412.592,Z 423.519,A -85,B 0,C 180,E1 -10544.048,E2 -10544.048} C_VEL
LIN {X 0,Y 413.529,Z 411.855,A -85,B 0,C 180,E1 -10545.147,E2 -10545.147} C_VEL
LIN {X 0,Y 414.385,Z 400.449,A -85,B 0,C 180,E1 -10545.998,E2 -10545.998} C_VEL
LIN {X 0,Y 413.783,Z 388.853,A -85,B 0,C 180,E1 -10546.719,E2 -10546.719} C_VEL
LIN {X 0,Y 412.37,Z 375.739,A -85,B 0,C 180,E1 -10547.368,E2 -10547.368} C_VEL
LIN {X 0,Y 410.432,Z 364.212,A -85,B 0,C 180,E1 -10547.813,E2 -10547.813} C_VEL
LIN {X 0,Y 410.792,Z 355.207,A -85,B 0,C 180,E1 -10551.056,E2 -10551.056} C_VEL
LIN {X 0,Y 411.112,Z 346.653,A -85,B 0,C 180,E1 -10554.223,E2 -10554.223} C_VEL
LIN {X 0,Y 411.663,Z 338.206,A -85,B 0,C 180,E1 -10557.449,E2 -10557.449} C_VEL
LIN {X 0,Y 412.295,Z 329.89,A -85,B 0,C 180,E1 -10560.756,E2 -10560.756} C_VEL
LIN {X 0,Y 412.889,Z 323.347,A -85,B 0,C 180,E1 -10563.482,E2 -10563.482} C_VEL
LIN {X 0,Y 413.488,Z 317.802,A -85,B 0,C 180,E1 -10565.902,E2 -10565.902} C_VEL
LIN {X 0,Y 413.154,Z 313.891,A -85,B 0,C 180,E1 -10567.762,E2 -10567.762} C_VEL
LIN {X 0,Y 411.946,Z 307.048,A -85,B 0,C 180,E1 -10571.352,E2 -10571.352} C_VEL
LIN {X 0,Y 411.185,Z 303.271,A -85,B 0,C 180,E1 -10573.606,E2 -10573.606} C_VEL
LIN {X 0,Y 411.177,Z 303.274,A -85,B 0,C 180,E1 -10576.867,E2 -10576.867} C_VEL
LIN {X 0,Y 411.219,Z 303.266,A -85,B 0,C 180,E1 -10580.272,E2 -10580.272} C_VEL
LIN {X 0,Y 411.197,Z 303.265,A -85,B 0,C 180,E1 -10583.447,E2 -10583.447} C_VEL
LIN {X 0,Y 411.211,Z 303.265,A -85,B 0,C 180,E1 -10586.873,E2 -10586.873} C_VEL
LIN {X 0,Y 411.237,Z 303.261,A -85,B 0,C 180,E1 -10590.644,E2 -10590.644} C_VEL
LIN {X 0,Y 411.243,Z 303.26,A -85,B 0,C 180,E1 -10593.619,E2 -10593.619} C_VEL
LIN {X 0,Y 411.208,Z 303.266,A -85,B 0,C 180,E1 -10596.853,E2 -10596.853} C_VEL
LIN {X 0,Y 411.219,Z 303.262,A -85,B 0,C 180,E1 -10600.05,E2 -10600.05} C_VEL
LIN {X 0,Y 411.268,Z 303.258,A -85,B 0,C 180,E1 -10603.131,E2 -10603.131} C_VEL
LIN {X 0,Y 411.31,Z 303.25,A -85,B 0,C 180,E1 -10606.896,E2 -10606.896} C_VEL
LIN {X 0,Y 411.296,Z 303.255,A -85,B 0,C 180,E1 -10610.161,E2 -10610.161} C_VEL
LIN {X 0,Y 411.427,Z 303.236,A -85,B 0,C 180,E1 -10613.132,E2 -10613.132} C_VEL
